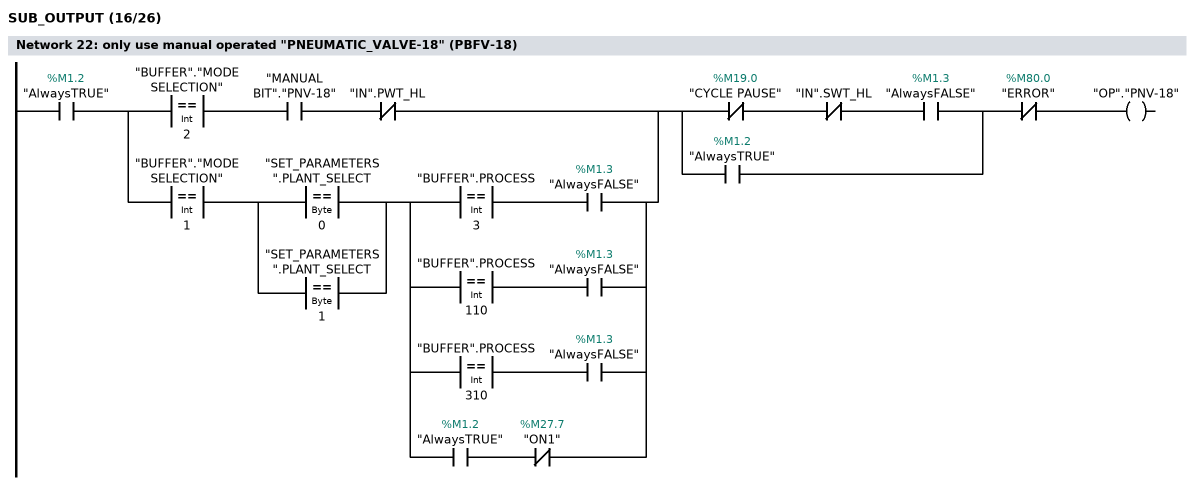
   RUNG wire#powerrail
      Contact( "AlwaysTRUE" )
      wire#w1
      { S7_Templates := "SrcType := Int" } EQ_Contact(in1 := "BUFFER"."MODE SELECTION", in2 := 2)
      Contact( "MANUAL BIT"."PNV-18" )
      I_Contact( "IN".PWT_HL )
      wire#w2
      I_Contact( "CYCLE PAUSE" )
      I_Contact( "IN".SWT_HL )
      Contact( "AlwaysFALSE" )
      wire#w5
      I_Contact( "ERROR" )
      Coil( "OP"."PNV-18" )
   END_RUNG
   RUNG wire#w1
      { S7_Templates := "SrcType := Int" } EQ_Contact(in1 := "BUFFER"."MODE SELECTION", in2 := 1)
      wire#w3
      { S7_Templates := "SrcType := Byte" } EQ_Contact(in1 := "SET_PARAMETERS".PLANT_SELECT, in2 := 0)
      wire#w4
      { S7_Templates := "SrcType := Int" } EQ_Contact(in1 := "BUFFER".PROCESS, in2 := 3)
      Contact( "AlwaysFALSE" )
   END_RUNG wire#w2
   RUNG wire#w3
      { S7_Templates := "SrcType := Byte" } EQ_Contact(in1 := "SET_PARAMETERS".PLANT_SELECT, in2 := 1)
   END_RUNG wire#w4
   RUNG wire#w4
      { S7_Templates := "SrcType := Int" } EQ_Contact(in1 := "BUFFER".PROCESS, in2 := 110)
      Contact( "AlwaysFALSE" )
   END_RUNG wire#w2
   RUNG wire#w4
      { S7_Templates := "SrcType := Int" } EQ_Contact(in1 := "BUFFER".PROCESS, in2 := 310)
      Contact( "AlwaysFALSE" )
   END_RUNG wire#w2
   RUNG wire#w4
      Contact( "AlwaysTRUE" )
      I_Contact( "ON1" )
   END_RUNG wire#w2
   RUNG wire#w2
      Contact( "AlwaysTRUE" )
   END_RUNG wire#w5
   // the same network as SCL:
   "OP"."PNV-18" := "AlwaysTRUE" AND ((("BUFFER"."MODE SELECTION" = 2) AND "MANUAL BIT"."PNV-18" AND NOT "IN".PWT_HL) OR (("BUFFER"."MODE SELECTION" = 1) AND (("SET_PARAMETERS".PLANT_SELECT = 0) OR ("SET_PARAMETERS".PLANT_SELECT = 1)) AND ((("BUFFER".PROCESS = 3) AND "AlwaysFALSE") OR (("BUFFER".PROCESS = 110) AND "AlwaysFALSE") OR (("BUFFER".PROCESS = 310) AND "AlwaysFALSE") OR ("AlwaysTRUE" AND NOT "ON1")))) AND ((NOT "CYCLE PAUSE" AND NOT "IN".SWT_HL AND "AlwaysFALSE") OR "AlwaysTRUE") AND NOT "ERROR";
END_REGION

REGION Network 23: "PNEUMATIC_VALVE-19" (PBFV-19) MFG2 - MFG
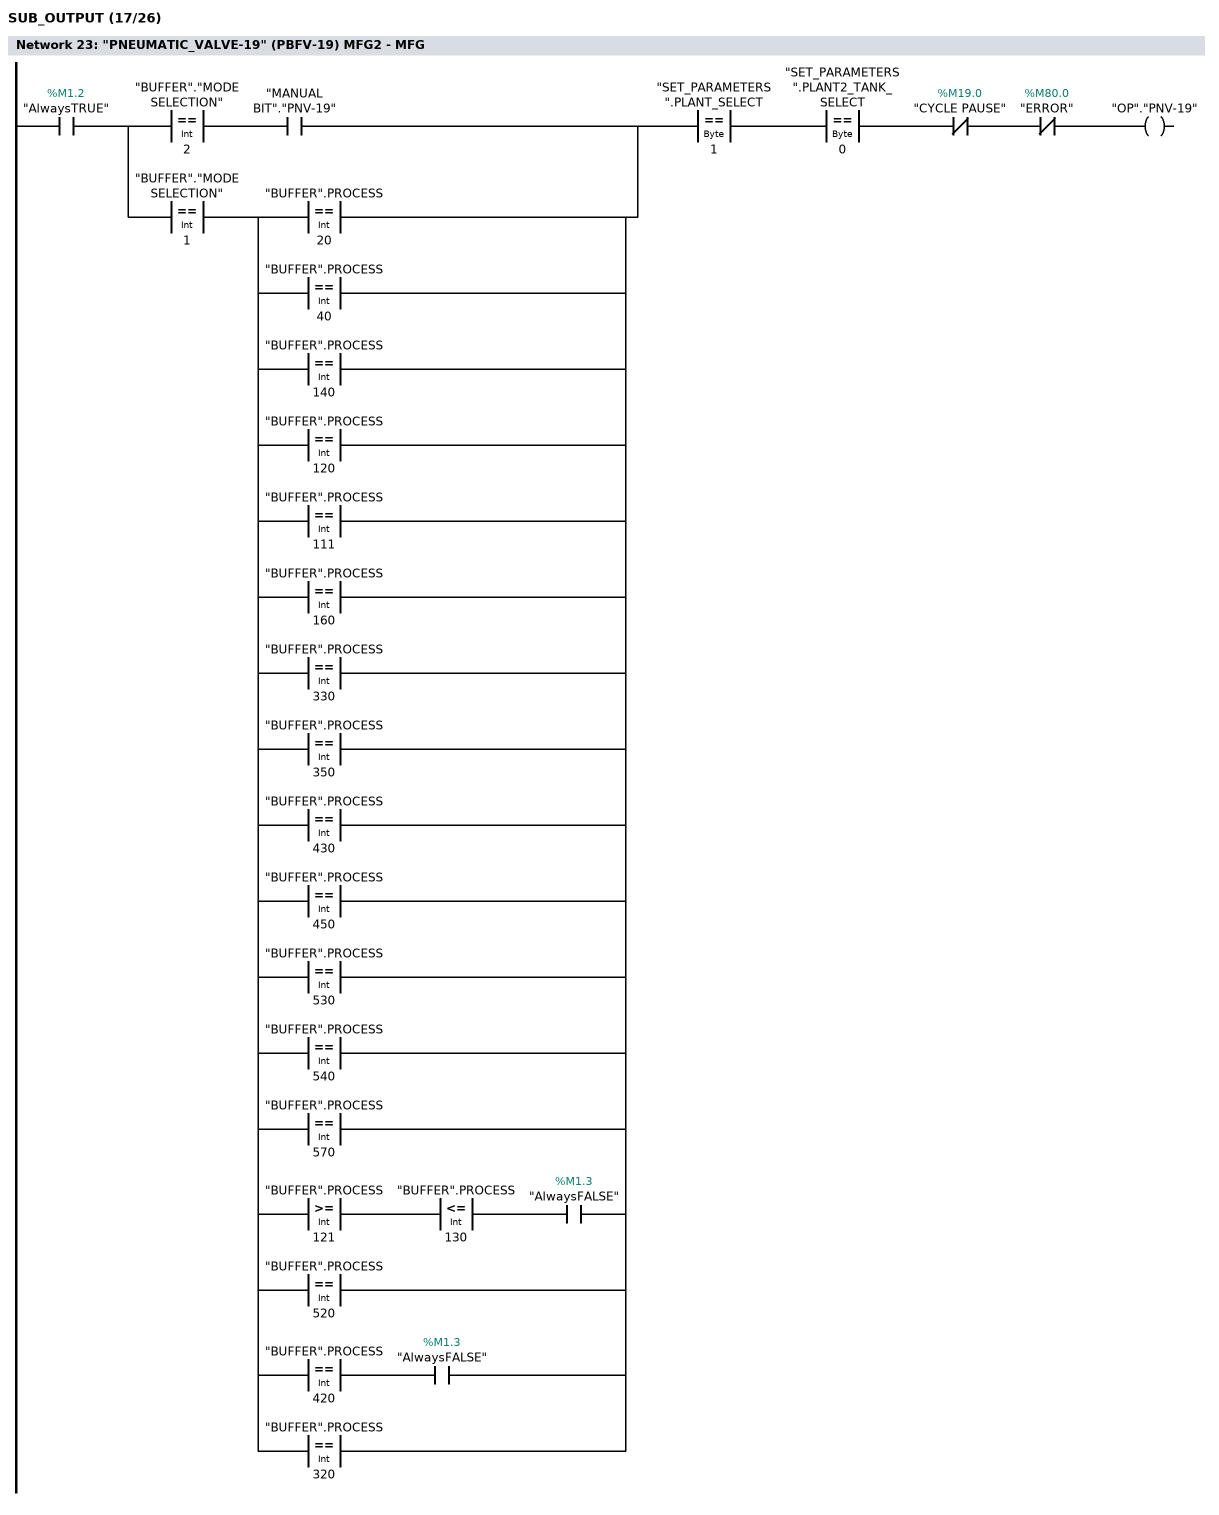
   RUNG wire#powerrail
      Contact( "AlwaysTRUE" )
      wire#w1
      { S7_Templates := "SrcType := Int" } EQ_Contact(in1 := "BUFFER"."MODE SELECTION", in2 := 2)
      Contact( "MANUAL BIT"."PNV-19" )
      wire#w2
      { S7_Templates := "SrcType := Byte" } EQ_Contact(in1 := "SET_PARAMETERS".PLANT_SELECT, in2 := 1)
      { S7_Templates := "SrcType := Byte" } EQ_Contact(in1 := "SET_PARAMETERS".PLANT2_TANK_SELECT, in2 := 0)
      I_Contact( "CYCLE PAUSE" )
      I_Contact( "ERROR" )
      Coil( "OP"."PNV-19" )
   END_RUNG
   RUNG wire#w1
      { S7_Templates := "SrcType := Int" } EQ_Contact(in1 := "BUFFER"."MODE SELECTION", in2 := 1)
      wire#w3
      { S7_Templates := "SrcType := Int" } EQ_Contact(in1 := "BUFFER".PROCESS, in2 := 20)
   END_RUNG wire#w2
   RUNG wire#w3
      { S7_Templates := "SrcType := Int" } EQ_Contact(in1 := "BUFFER".PROCESS, in2 := 40)
   END_RUNG wire#w2
   RUNG wire#w3
      { S7_Templates := "SrcType := Int" } EQ_Contact(in1 := "BUFFER".PROCESS, in2 := 140)
   END_RUNG wire#w2
   RUNG wire#w3
      { S7_Templates := "SrcType := Int" } EQ_Contact(in1 := "BUFFER".PROCESS, in2 := 120)
   END_RUNG wire#w2
   RUNG wire#w3
      { S7_Templates := "SrcType := Int" } EQ_Contact(in1 := "BUFFER".PROCESS, in2 := 111)
   END_RUNG wire#w2
   RUNG wire#w3
      { S7_Templates := "SrcType := Int" } EQ_Contact(in1 := "BUFFER".PROCESS, in2 := 160)
   END_RUNG wire#w2
   RUNG wire#w3
      { S7_Templates := "SrcType := Int" } EQ_Contact(in1 := "BUFFER".PROCESS, in2 := 330)
   END_RUNG wire#w2
   RUNG wire#w3
      { S7_Templates := "SrcType := Int" } EQ_Contact(in1 := "BUFFER".PROCESS, in2 := 350)
   END_RUNG wire#w2
   RUNG wire#w3
      { S7_Templates := "SrcType := Int" } EQ_Contact(in1 := "BUFFER".PROCESS, in2 := 430)
   END_RUNG wire#w2
   RUNG wire#w3
      { S7_Templates := "SrcType := Int" } EQ_Contact(in1 := "BUFFER".PROCESS, in2 := 450)
   END_RUNG wire#w2
   RUNG wire#w3
      { S7_Templates := "SrcType := Int" } EQ_Contact(in1 := "BUFFER".PROCESS, in2 := 530)
   END_RUNG wire#w2
   RUNG wire#w3
      { S7_Templates := "SrcType := Int" } EQ_Contact(in1 := "BUFFER".PROCESS, in2 := 540)
   END_RUNG wire#w2
   RUNG wire#w3
      { S7_Templates := "SrcType := Int" } EQ_Contact(in1 := "BUFFER".PROCESS, in2 := 570)
   END_RUNG wire#w2
   RUNG wire#w3
      { S7_Templates := "SrcType := Int" } GE_Contact(in1 := "BUFFER".PROCESS, in2 := 121)
      { S7_Templates := "SrcType := Int" } LE_Contact(in1 := "BUFFER".PROCESS, in2 := 130)
      Contact( "AlwaysFALSE" )
   END_RUNG wire#w2
   RUNG wire#w3
      { S7_Templates := "SrcType := Int" } EQ_Contact(in1 := "BUFFER".PROCESS, in2 := 520)
   END_RUNG wire#w2
   RUNG wire#w3
      { S7_Templates := "SrcType := Int" } EQ_Contact(in1 := "BUFFER".PROCESS, in2 := 420)
      Contact( "AlwaysFALSE" )
   END_RUNG wire#w2
   RUNG wire#w3
      { S7_Templates := "SrcType := Int" } EQ_Contact(in1 := "BUFFER".PROCESS, in2 := 320)
   END_RUNG wire#w2
   // the same network as SCL:
   "OP"."PNV-19" := "AlwaysTRUE" AND ((("BUFFER"."MODE SELECTION" = 2) AND "MANUAL BIT"."PNV-19") OR (("BUFFER"."MODE SELECTION" = 1) AND (("BUFFER".PROCESS = 20) OR ("BUFFER".PROCESS = 40) OR ("BUFFER".PROCESS = 140) OR ("BUFFER".PROCESS = 120) OR ("BUFFER".PROCESS = 111) OR ("BUFFER".PROCESS = 160) OR ("BUFFER".PROCESS = 330) OR ("BUFFER".PROCESS = 350) OR ("BUFFER".PROCESS = 430) OR ("BUFFER".PROCESS = 450) OR ("BUFFER".PROCESS = 530) OR ("BUFFER".PROCESS = 540) OR ("BUFFER".PROCESS = 570) OR (("BUFFER".PROCESS >= 121) AND ("BUFFER".PROCESS <= 130) AND "AlwaysFALSE") OR ("BUFFER".PROCESS = 520) OR (("BUFFER".PROCESS = 420) AND "AlwaysFALSE") OR ("BUFFER".PROCESS = 320)))) AND ("SET_PARAMETERS".PLANT_SELECT = 1) AND ("SET_PARAMETERS".PLANT2_TANK_SELECT = 0) AND NOT "CYCLE PAUSE" AND NOT "ERROR";
END_REGION

REGION Network 24: "PNEUMATIC_VALVE-20" (PBFV-20) MFG2- STORAGE1
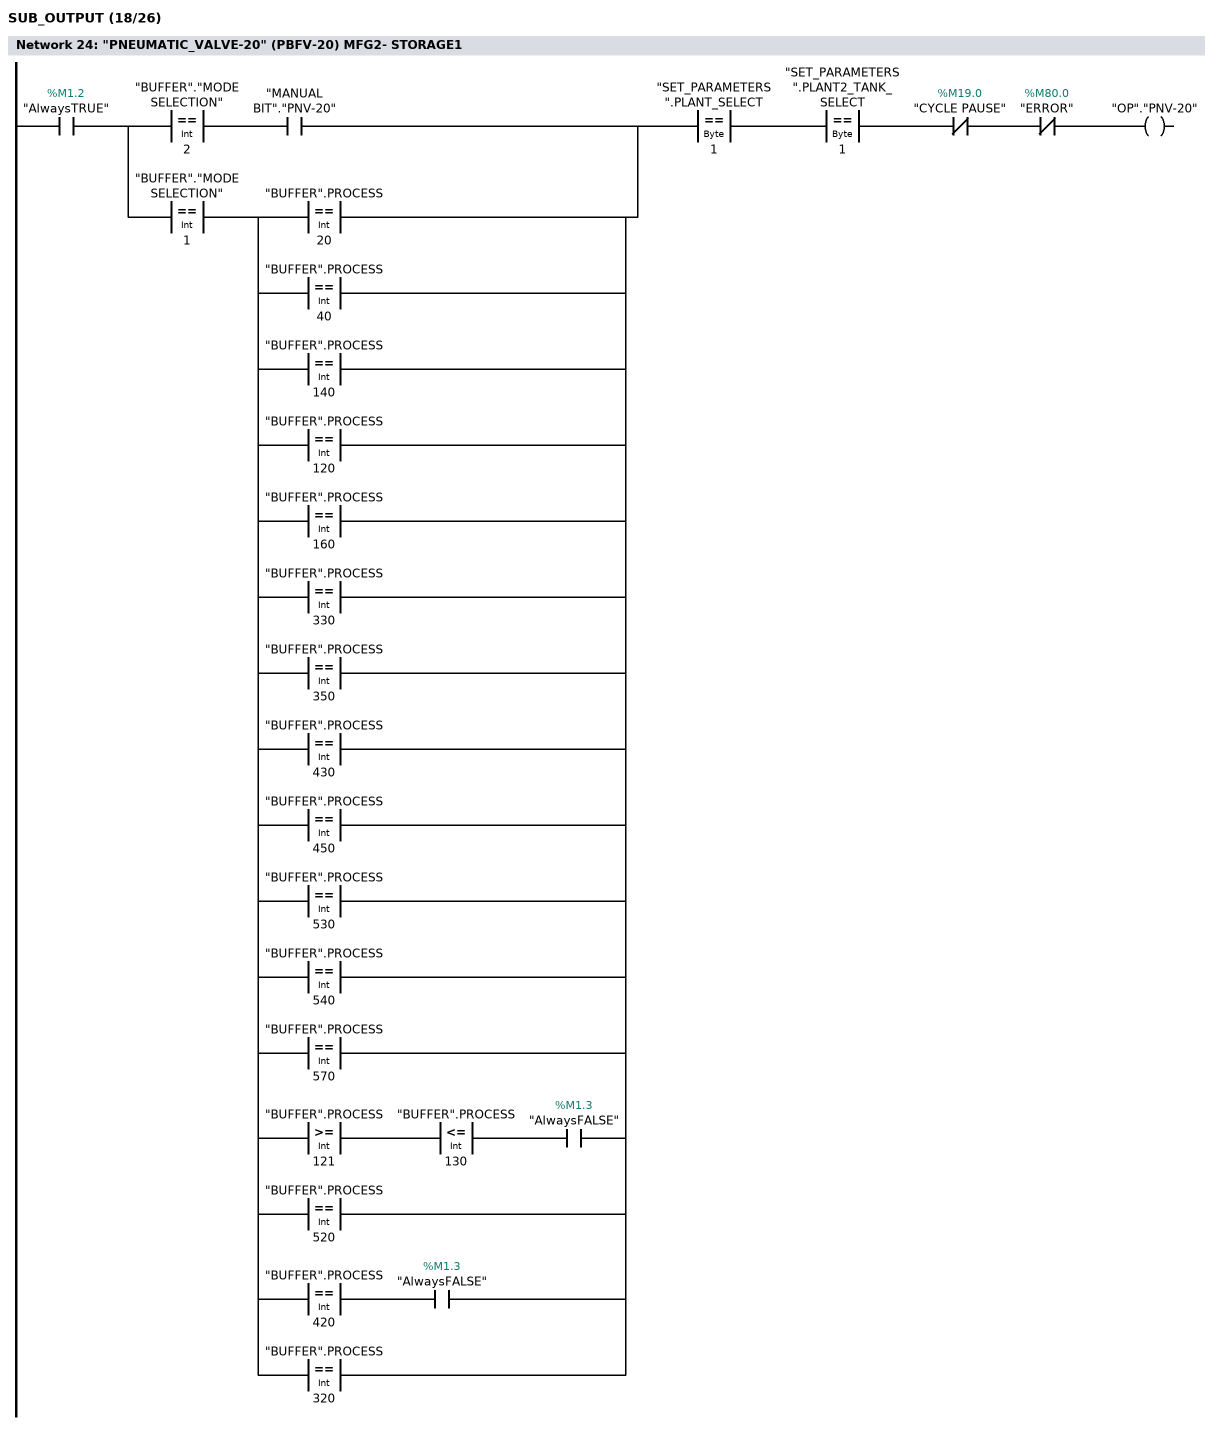
   RUNG wire#powerrail
      Contact( "AlwaysTRUE" )
      wire#w1
      { S7_Templates := "SrcType := Int" } EQ_Contact(in1 := "BUFFER"."MODE SELECTION", in2 := 2)
      Contact( "MANUAL BIT"."PNV-20" )
      wire#w2
      { S7_Templates := "SrcType := Byte" } EQ_Contact(in1 := "SET_PARAMETERS".PLANT_SELECT, in2 := 1)
      { S7_Templates := "SrcType := Byte" } EQ_Contact(in1 := "SET_PARAMETERS".PLANT2_TANK_SELECT, in2 := 1)
      I_Contact( "CYCLE PAUSE" )
      I_Contact( "ERROR" )
      Coil( "OP"."PNV-20" )
   END_RUNG
   RUNG wire#w1
      { S7_Templates := "SrcType := Int" } EQ_Contact(in1 := "BUFFER"."MODE SELECTION", in2 := 1)
      wire#w3
      { S7_Templates := "SrcType := Int" } EQ_Contact(in1 := "BUFFER".PROCESS, in2 := 20)
   END_RUNG wire#w2
   RUNG wire#w3
      { S7_Templates := "SrcType := Int" } EQ_Contact(in1 := "BUFFER".PROCESS, in2 := 40)
   END_RUNG wire#w2
   RUNG wire#w3
      { S7_Templates := "SrcType := Int" } EQ_Contact(in1 := "BUFFER".PROCESS, in2 := 140)
   END_RUNG wire#w2
   RUNG wire#w3
      { S7_Templates := "SrcType := Int" } EQ_Contact(in1 := "BUFFER".PROCESS, in2 := 120)
   END_RUNG wire#w2
   RUNG wire#w3
      { S7_Templates := "SrcType := Int" } EQ_Contact(in1 := "BUFFER".PROCESS, in2 := 160)
   END_RUNG wire#w2
   RUNG wire#w3
      { S7_Templates := "SrcType := Int" } EQ_Contact(in1 := "BUFFER".PROCESS, in2 := 330)
   END_RUNG wire#w2
   RUNG wire#w3
      { S7_Templates := "SrcType := Int" } EQ_Contact(in1 := "BUFFER".PROCESS, in2 := 350)
   END_RUNG wire#w2
   RUNG wire#w3
      { S7_Templates := "SrcType := Int" } EQ_Contact(in1 := "BUFFER".PROCESS, in2 := 430)
   END_RUNG wire#w2
   RUNG wire#w3
      { S7_Templates := "SrcType := Int" } EQ_Contact(in1 := "BUFFER".PROCESS, in2 := 450)
   END_RUNG wire#w2
   RUNG wire#w3
      { S7_Templates := "SrcType := Int" } EQ_Contact(in1 := "BUFFER".PROCESS, in2 := 530)
   END_RUNG wire#w2
   RUNG wire#w3
      { S7_Templates := "SrcType := Int" } EQ_Contact(in1 := "BUFFER".PROCESS, in2 := 540)
   END_RUNG wire#w2
   RUNG wire#w3
      { S7_Templates := "SrcType := Int" } EQ_Contact(in1 := "BUFFER".PROCESS, in2 := 570)
   END_RUNG wire#w2
   RUNG wire#w3
      { S7_Templates := "SrcType := Int" } GE_Contact(in1 := "BUFFER".PROCESS, in2 := 121)
      { S7_Templates := "SrcType := Int" } LE_Contact(in1 := "BUFFER".PROCESS, in2 := 130)
      Contact( "AlwaysFALSE" )
   END_RUNG wire#w2
   RUNG wire#w3
      { S7_Templates := "SrcType := Int" } EQ_Contact(in1 := "BUFFER".PROCESS, in2 := 520)
   END_RUNG wire#w2
   RUNG wire#w3
      { S7_Templates := "SrcType := Int" } EQ_Contact(in1 := "BUFFER".PROCESS, in2 := 420)
      Contact( "AlwaysFALSE" )
   END_RUNG wire#w2
   RUNG wire#w3
      { S7_Templates := "SrcType := Int" } EQ_Contact(in1 := "BUFFER".PROCESS, in2 := 320)
   END_RUNG wire#w2
   // the same network as SCL:
   "OP"."PNV-20" := "AlwaysTRUE" AND ((("BUFFER"."MODE SELECTION" = 2) AND "MANUAL BIT"."PNV-20") OR (("BUFFER"."MODE SELECTION" = 1) AND (("BUFFER".PROCESS = 20) OR ("BUFFER".PROCESS = 40) OR ("BUFFER".PROCESS = 140) OR ("BUFFER".PROCESS = 120) OR ("BUFFER".PROCESS = 160) OR ("BUFFER".PROCESS = 330) OR ("BUFFER".PROCESS = 350) OR ("BUFFER".PROCESS = 430) OR ("BUFFER".PROCESS = 450) OR ("BUFFER".PROCESS = 530) OR ("BUFFER".PROCESS = 540) OR ("BUFFER".PROCESS = 570) OR (("BUFFER".PROCESS >= 121) AND ("BUFFER".PROCESS <= 130) AND "AlwaysFALSE") OR ("BUFFER".PROCESS = 520) OR (("BUFFER".PROCESS = 420) AND "AlwaysFALSE") OR ("BUFFER".PROCESS = 320)))) AND ("SET_PARAMETERS".PLANT_SELECT = 1) AND ("SET_PARAMETERS".PLANT2_TANK_SELECT = 1) AND NOT "CYCLE PAUSE" AND NOT "ERROR";
END_REGION

REGION Network 25: "PNEUMATIC_VALVE-21" (PV-21)
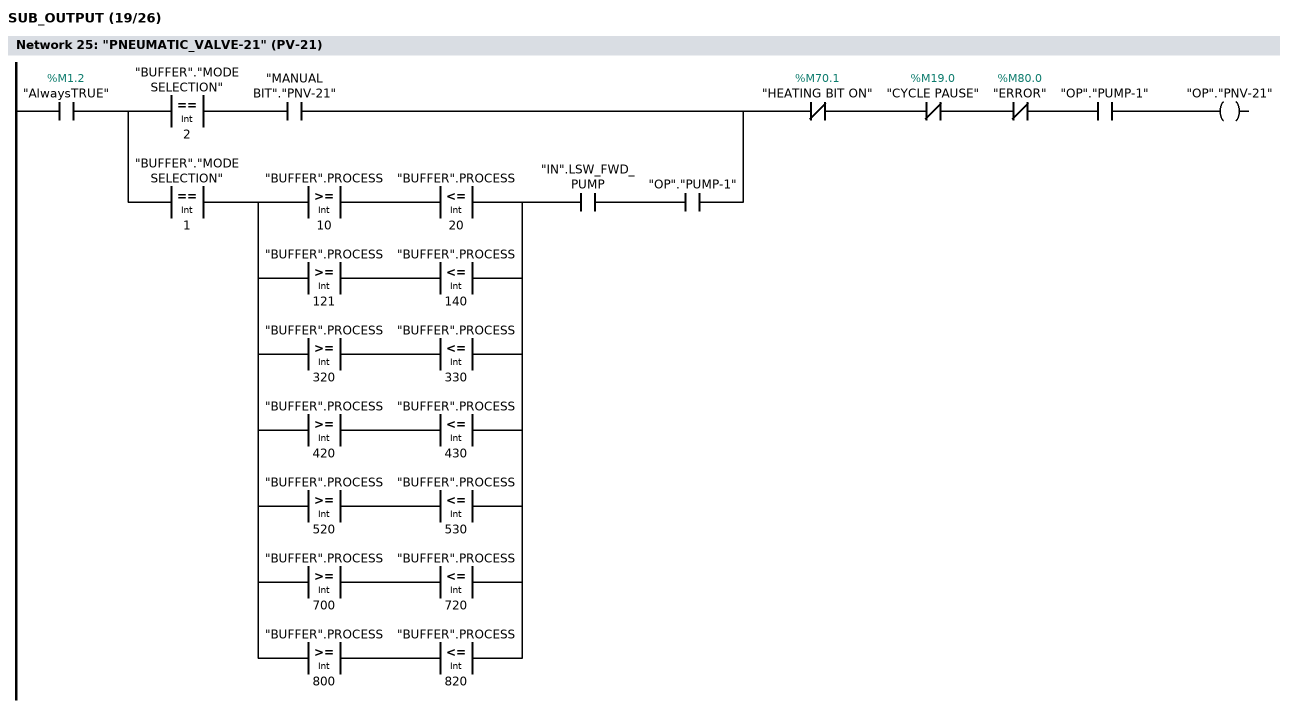
   RUNG wire#powerrail
      Contact( "AlwaysTRUE" )
      wire#w1
      { S7_Templates := "SrcType := Int" } EQ_Contact(in1 := "BUFFER"."MODE SELECTION", in2 := 2)
      Contact( "MANUAL BIT"."PNV-21" )
      wire#w2
      I_Contact( "HEATING BIT ON" )
      I_Contact( "CYCLE PAUSE" )
      I_Contact( "ERROR" )
      Contact( "OP"."PUMP-1" )
      Coil( "OP"."PNV-21" )
   END_RUNG
   RUNG wire#w1
      { S7_Templates := "SrcType := Int" } EQ_Contact(in1 := "BUFFER"."MODE SELECTION", in2 := 1)
      wire#w3
      { S7_Templates := "SrcType := Int" } GE_Contact(in1 := "BUFFER".PROCESS, in2 := 10)
      { S7_Templates := "SrcType := Int" } LE_Contact(in1 := "BUFFER".PROCESS, in2 := 20)
      wire#w4
      Contact( "IN".LSW_FWD_PUMP )
      Contact( "OP"."PUMP-1" )
   END_RUNG wire#w2
   RUNG wire#w3
      { S7_Templates := "SrcType := Int" } GE_Contact(in1 := "BUFFER".PROCESS, in2 := 121)
      { S7_Templates := "SrcType := Int" } LE_Contact(in1 := "BUFFER".PROCESS, in2 := 140)
   END_RUNG wire#w4
   RUNG wire#w3
      { S7_Templates := "SrcType := Int" } GE_Contact(in1 := "BUFFER".PROCESS, in2 := 320)
      { S7_Templates := "SrcType := Int" } LE_Contact(in1 := "BUFFER".PROCESS, in2 := 330)
   END_RUNG wire#w4
   RUNG wire#w3
      { S7_Templates := "SrcType := Int" } GE_Contact(in1 := "BUFFER".PROCESS, in2 := 420)
      { S7_Templates := "SrcType := Int" } LE_Contact(in1 := "BUFFER".PROCESS, in2 := 430)
   END_RUNG wire#w4
   RUNG wire#w3
      { S7_Templates := "SrcType := Int" } GE_Contact(in1 := "BUFFER".PROCESS, in2 := 520)
      { S7_Templates := "SrcType := Int" } LE_Contact(in1 := "BUFFER".PROCESS, in2 := 530)
   END_RUNG wire#w4
   RUNG wire#w3
      { S7_Templates := "SrcType := Int" } GE_Contact(in1 := "BUFFER".PROCESS, in2 := 700)
      { S7_Templates := "SrcType := Int" } LE_Contact(in1 := "BUFFER".PROCESS, in2 := 720)
   END_RUNG wire#w4
   RUNG wire#w3
      { S7_Templates := "SrcType := Int" } GE_Contact(in1 := "BUFFER".PROCESS, in2 := 800)
      { S7_Templates := "SrcType := Int" } LE_Contact(in1 := "BUFFER".PROCESS, in2 := 820)
   END_RUNG wire#w4
   // the same network as SCL:
   "OP"."PNV-21" := "AlwaysTRUE" AND ((("BUFFER"."MODE SELECTION" = 2) AND "MANUAL BIT"."PNV-21") OR (("BUFFER"."MODE SELECTION" = 1) AND ((("BUFFER".PROCESS >= 10) AND ("BUFFER".PROCESS <= 20)) OR (("BUFFER".PROCESS >= 121) AND ("BUFFER".PROCESS <= 140)) OR (("BUFFER".PROCESS >= 320) AND ("BUFFER".PROCESS <= 330)) OR (("BUFFER".PROCESS >= 420) AND ("BUFFER".PROCESS <= 430)) OR (("BUFFER".PROCESS >= 520) AND ("BUFFER".PROCESS <= 530)) OR (("BUFFER".PROCESS >= 700) AND ("BUFFER".PROCESS <= 720)) OR (("BUFFER".PROCESS >= 800) AND ("BUFFER".PROCESS <= 820))) AND "IN".LSW_FWD_PUMP AND "OP"."PUMP-1")) AND NOT "HEATING BIT ON" AND NOT "CYCLE PAUSE" AND NOT "ERROR" AND "OP"."PUMP-1";
END_REGION

REGION Network 26: "PNEUMATIC_VALVE-22" (PV-22)
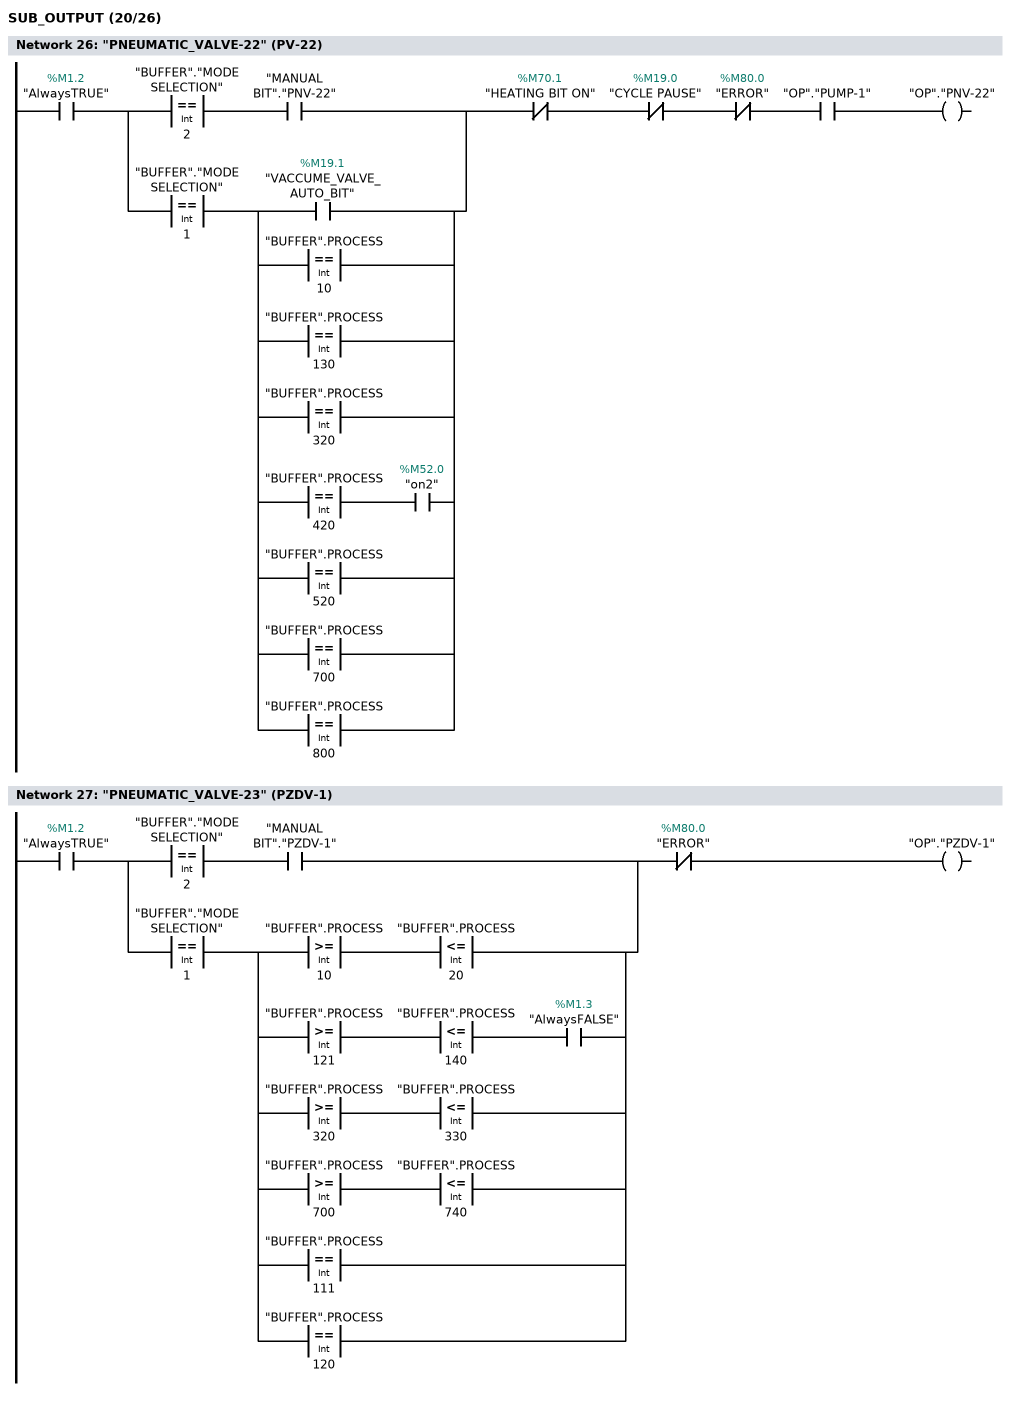
   RUNG wire#powerrail
      Contact( "AlwaysTRUE" )
      wire#w1
      { S7_Templates := "SrcType := Int" } EQ_Contact(in1 := "BUFFER"."MODE SELECTION", in2 := 2)
      Contact( "MANUAL BIT"."PNV-22" )
      wire#w2
      I_Contact( "HEATING BIT ON" )
      I_Contact( "CYCLE PAUSE" )
      I_Contact( "ERROR" )
      Contact( "OP"."PUMP-1" )
      Coil( "OP"."PNV-22" )
   END_RUNG
   RUNG wire#w1
      { S7_Templates := "SrcType := Int" } EQ_Contact(in1 := "BUFFER"."MODE SELECTION", in2 := 1)
      wire#w3
      Contact( "VACCUME_VALVE_AUTO_BIT" )
   END_RUNG wire#w2
   RUNG wire#w3
      { S7_Templates := "SrcType := Int" } EQ_Contact(in1 := "BUFFER".PROCESS, in2 := 10)
   END_RUNG wire#w2
   RUNG wire#w3
      { S7_Templates := "SrcType := Int" } EQ_Contact(in1 := "BUFFER".PROCESS, in2 := 130)
   END_RUNG wire#w2
   RUNG wire#w3
      { S7_Templates := "SrcType := Int" } EQ_Contact(in1 := "BUFFER".PROCESS, in2 := 320)
   END_RUNG wire#w2
   RUNG wire#w3
      { S7_Templates := "SrcType := Int" } EQ_Contact(in1 := "BUFFER".PROCESS, in2 := 420)
      Contact( "on2" )
   END_RUNG wire#w2
   RUNG wire#w3
      { S7_Templates := "SrcType := Int" } EQ_Contact(in1 := "BUFFER".PROCESS, in2 := 520)
   END_RUNG wire#w2
   RUNG wire#w3
      { S7_Templates := "SrcType := Int" } EQ_Contact(in1 := "BUFFER".PROCESS, in2 := 700)
   END_RUNG wire#w2
   RUNG wire#w3
      { S7_Templates := "SrcType := Int" } EQ_Contact(in1 := "BUFFER".PROCESS, in2 := 800)
   END_RUNG wire#w2
   // the same network as SCL:
   "OP"."PNV-22" := "AlwaysTRUE" AND ((("BUFFER"."MODE SELECTION" = 2) AND "MANUAL BIT"."PNV-22") OR (("BUFFER"."MODE SELECTION" = 1) AND ("VACCUME_VALVE_AUTO_BIT" OR ("BUFFER".PROCESS = 10) OR ("BUFFER".PROCESS = 130) OR ("BUFFER".PROCESS = 320) OR (("BUFFER".PROCESS = 420) AND "on2") OR ("BUFFER".PROCESS = 520) OR ("BUFFER".PROCESS = 700) OR ("BUFFER".PROCESS = 800)))) AND NOT "HEATING BIT ON" AND NOT "CYCLE PAUSE" AND NOT "ERROR" AND "OP"."PUMP-1";
END_REGION

REGION Network 27: "PNEUMATIC_VALVE-23" (PZDV-1)
   RUNG wire#powerrail
      Contact( "AlwaysTRUE" )
      wire#w1
      { S7_Templates := "SrcType := Int" } EQ_Contact(in1 := "BUFFER"."MODE SELECTION", in2 := 2)
      Contact( "MANUAL BIT"."PZDV-1" )
      wire#w2
      I_Contact( "ERROR" )
      Coil( "OP"."PZDV-1" )
   END_RUNG
   RUNG wire#w1
      { S7_Templates := "SrcType := Int" } EQ_Contact(in1 := "BUFFER"."MODE SELECTION", in2 := 1)
      wire#w3
      { S7_Templates := "SrcType := Int" } GE_Contact(in1 := "BUFFER".PROCESS, in2 := 10)
      { S7_Templates := "SrcType := Int" } LE_Contact(in1 := "BUFFER".PROCESS, in2 := 20)
   END_RUNG wire#w2
   RUNG wire#w3
      { S7_Templates := "SrcType := Int" } GE_Contact(in1 := "BUFFER".PROCESS, in2 := 121)
      { S7_Templates := "SrcType := Int" } LE_Contact(in1 := "BUFFER".PROCESS, in2 := 140)
      Contact( "AlwaysFALSE" )
   END_RUNG wire#w2
   RUNG wire#w3
      { S7_Templates := "SrcType := Int" } GE_Contact(in1 := "BUFFER".PROCESS, in2 := 320)
      { S7_Templates := "SrcType := Int" } LE_Contact(in1 := "BUFFER".PROCESS, in2 := 330)
   END_RUNG wire#w2
   RUNG wire#w3
      { S7_Templates := "SrcType := Int" } GE_Contact(in1 := "BUFFER".PROCESS, in2 := 700)
      { S7_Templates := "SrcType := Int" } LE_Contact(in1 := "BUFFER".PROCESS, in2 := 740)
   END_RUNG wire#w2
   RUNG wire#w3
      { S7_Templates := "SrcType := Int" } EQ_Contact(in1 := "BUFFER".PROCESS, in2 := 111)
   END_RUNG wire#w2
   RUNG wire#w3
      { S7_Templates := "SrcType := Int" } EQ_Contact(in1 := "BUFFER".PROCESS, in2 := 120)
   END_RUNG wire#w2
   // the same network as SCL:
   "OP"."PZDV-1" := "AlwaysTRUE" AND ((("BUFFER"."MODE SELECTION" = 2) AND "MANUAL BIT"."PZDV-1") OR (("BUFFER"."MODE SELECTION" = 1) AND ((("BUFFER".PROCESS >= 10) AND ("BUFFER".PROCESS <= 20)) OR (("BUFFER".PROCESS >= 121) AND ("BUFFER".PROCESS <= 140) AND "AlwaysFALSE") OR (("BUFFER".PROCESS >= 320) AND ("BUFFER".PROCESS <= 330)) OR (("BUFFER".PROCESS >= 700) AND ("BUFFER".PROCESS <= 740)) OR ("BUFFER".PROCESS = 111) OR ("BUFFER".PROCESS = 120)))) AND NOT "ERROR";
END_REGION

REGION Network 28: "PNEUMATIC_VALVE-24" (PZDV-2)
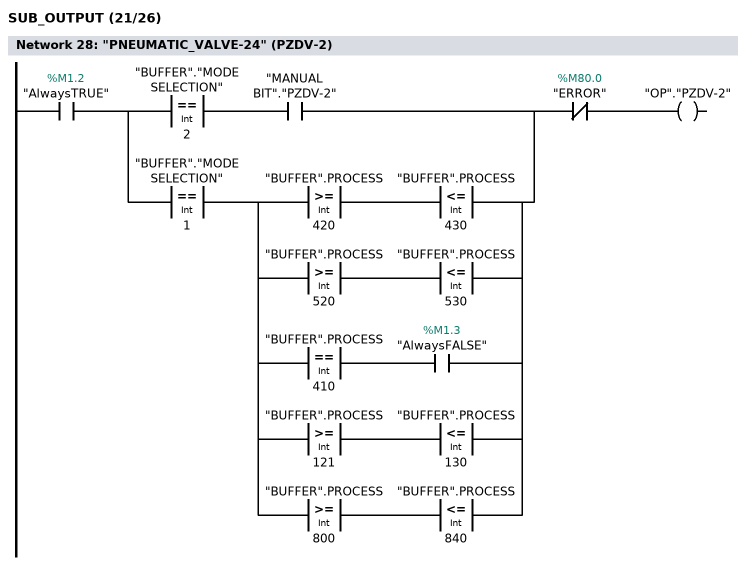
   RUNG wire#powerrail
      Contact( "AlwaysTRUE" )
      wire#w1
      { S7_Templates := "SrcType := Int" } EQ_Contact(in1 := "BUFFER"."MODE SELECTION", in2 := 2)
      Contact( "MANUAL BIT"."PZDV-2" )
      wire#w2
      I_Contact( "ERROR" )
      Coil( "OP"."PZDV-2" )
   END_RUNG
   RUNG wire#w1
      { S7_Templates := "SrcType := Int" } EQ_Contact(in1 := "BUFFER"."MODE SELECTION", in2 := 1)
      wire#w3
      { S7_Templates := "SrcType := Int" } GE_Contact(in1 := "BUFFER".PROCESS, in2 := 420)
      { S7_Templates := "SrcType := Int" } LE_Contact(in1 := "BUFFER".PROCESS, in2 := 430)
   END_RUNG wire#w2
   RUNG wire#w3
      { S7_Templates := "SrcType := Int" } GE_Contact(in1 := "BUFFER".PROCESS, in2 := 520)
      { S7_Templates := "SrcType := Int" } LE_Contact(in1 := "BUFFER".PROCESS, in2 := 530)
   END_RUNG wire#w2
   RUNG wire#w3
      { S7_Templates := "SrcType := Int" } EQ_Contact(in1 := "BUFFER".PROCESS, in2 := 410)
      Contact( "AlwaysFALSE" )
   END_RUNG wire#w2
   RUNG wire#w3
      { S7_Templates := "SrcType := Int" } GE_Contact(in1 := "BUFFER".PROCESS, in2 := 121)
      { S7_Templates := "SrcType := Int" } LE_Contact(in1 := "BUFFER".PROCESS, in2 := 130)
   END_RUNG wire#w2
   RUNG wire#w3
      { S7_Templates := "SrcType := Int" } GE_Contact(in1 := "BUFFER".PROCESS, in2 := 800)
      { S7_Templates := "SrcType := Int" } LE_Contact(in1 := "BUFFER".PROCESS, in2 := 840)
   END_RUNG wire#w2
   // the same network as SCL:
   "OP"."PZDV-2" := "AlwaysTRUE" AND ((("BUFFER"."MODE SELECTION" = 2) AND "MANUAL BIT"."PZDV-2") OR (("BUFFER"."MODE SELECTION" = 1) AND ((("BUFFER".PROCESS >= 420) AND ("BUFFER".PROCESS <= 430)) OR (("BUFFER".PROCESS >= 520) AND ("BUFFER".PROCESS <= 530)) OR (("BUFFER".PROCESS = 410) AND "AlwaysFALSE") OR (("BUFFER".PROCESS >= 121) AND ("BUFFER".PROCESS <= 130)) OR (("BUFFER".PROCESS >= 800) AND ("BUFFER".PROCESS <= 840))))) AND NOT "ERROR";
END_REGION

REGION Network 29: "PNEUMATIC_VALVE-25" (CIP_IN) MFG2- STORAGE2 PBFV-23
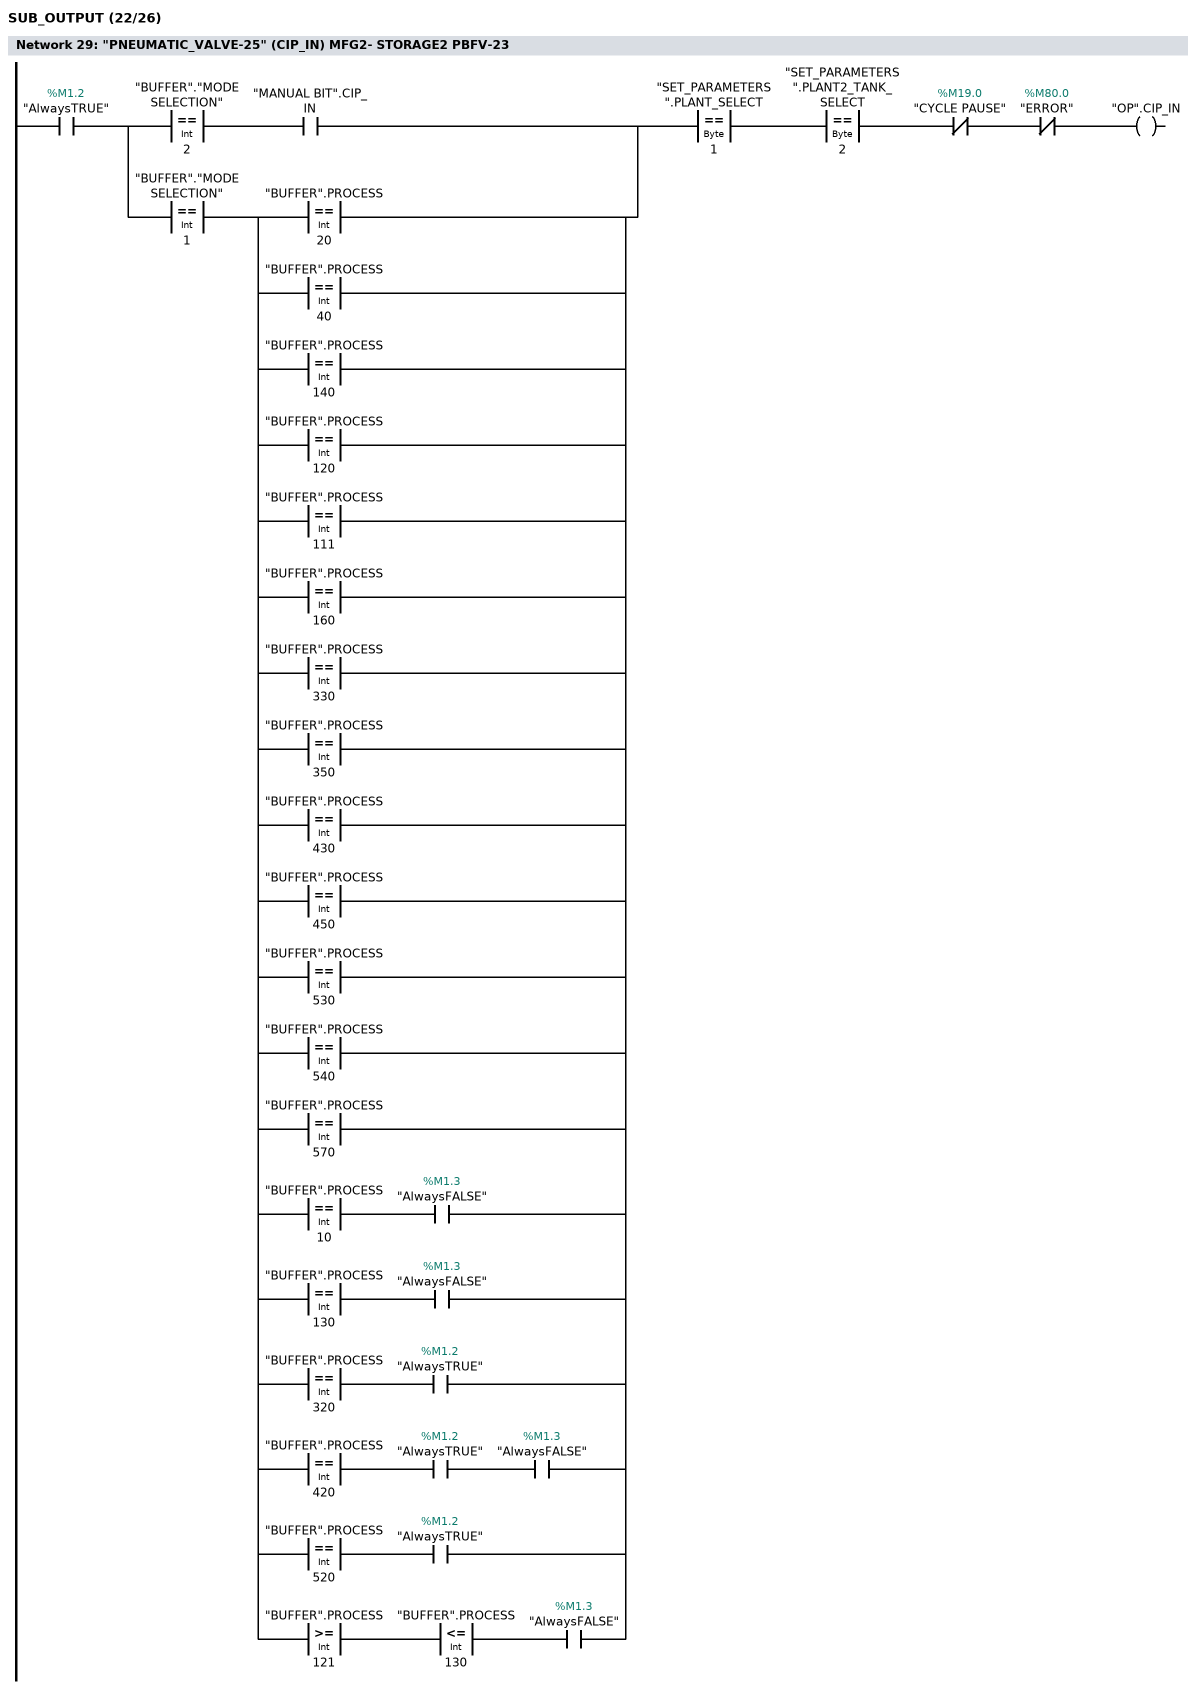
   RUNG wire#powerrail
      Contact( "AlwaysTRUE" )
      wire#w1
      { S7_Templates := "SrcType := Int" } EQ_Contact(in1 := "BUFFER"."MODE SELECTION", in2 := 2)
      Contact( "MANUAL BIT".CIP_IN )
      wire#w2
      { S7_Templates := "SrcType := Byte" } EQ_Contact(in1 := "SET_PARAMETERS".PLANT_SELECT, in2 := 1)
      { S7_Templates := "SrcType := Byte" } EQ_Contact(in1 := "SET_PARAMETERS".PLANT2_TANK_SELECT, in2 := 2)
      I_Contact( "CYCLE PAUSE" )
      I_Contact( "ERROR" )
      Coil( "OP".CIP_IN )
   END_RUNG
   RUNG wire#w1
      { S7_Templates := "SrcType := Int" } EQ_Contact(in1 := "BUFFER"."MODE SELECTION", in2 := 1)
      wire#w3
      { S7_Templates := "SrcType := Int" } EQ_Contact(in1 := "BUFFER".PROCESS, in2 := 20)
   END_RUNG wire#w2
   RUNG wire#w3
      { S7_Templates := "SrcType := Int" } EQ_Contact(in1 := "BUFFER".PROCESS, in2 := 40)
   END_RUNG wire#w2
   RUNG wire#w3
      { S7_Templates := "SrcType := Int" } EQ_Contact(in1 := "BUFFER".PROCESS, in2 := 140)
   END_RUNG wire#w2
   RUNG wire#w3
      { S7_Templates := "SrcType := Int" } EQ_Contact(in1 := "BUFFER".PROCESS, in2 := 120)
   END_RUNG wire#w2
   RUNG wire#w3
      { S7_Templates := "SrcType := Int" } EQ_Contact(in1 := "BUFFER".PROCESS, in2 := 111)
   END_RUNG wire#w2
   RUNG wire#w3
      { S7_Templates := "SrcType := Int" } EQ_Contact(in1 := "BUFFER".PROCESS, in2 := 160)
   END_RUNG wire#w2
   RUNG wire#w3
      { S7_Templates := "SrcType := Int" } EQ_Contact(in1 := "BUFFER".PROCESS, in2 := 330)
   END_RUNG wire#w2
   RUNG wire#w3
      { S7_Templates := "SrcType := Int" } EQ_Contact(in1 := "BUFFER".PROCESS, in2 := 350)
   END_RUNG wire#w2
   RUNG wire#w3
      { S7_Templates := "SrcType := Int" } EQ_Contact(in1 := "BUFFER".PROCESS, in2 := 430)
   END_RUNG wire#w2
   RUNG wire#w3
      { S7_Templates := "SrcType := Int" } EQ_Contact(in1 := "BUFFER".PROCESS, in2 := 450)
   END_RUNG wire#w2
   RUNG wire#w3
      { S7_Templates := "SrcType := Int" } EQ_Contact(in1 := "BUFFER".PROCESS, in2 := 530)
   END_RUNG wire#w2
   RUNG wire#w3
      { S7_Templates := "SrcType := Int" } EQ_Contact(in1 := "BUFFER".PROCESS, in2 := 540)
   END_RUNG wire#w2
   RUNG wire#w3
      { S7_Templates := "SrcType := Int" } EQ_Contact(in1 := "BUFFER".PROCESS, in2 := 570)
   END_RUNG wire#w2
   RUNG wire#w3
      { S7_Templates := "SrcType := Int" } EQ_Contact(in1 := "BUFFER".PROCESS, in2 := 10)
      Contact( "AlwaysFALSE" )
   END_RUNG wire#w2
   RUNG wire#w3
      { S7_Templates := "SrcType := Int" } EQ_Contact(in1 := "BUFFER".PROCESS, in2 := 130)
      Contact( "AlwaysFALSE" )
   END_RUNG wire#w2
   RUNG wire#w3
      { S7_Templates := "SrcType := Int" } EQ_Contact(in1 := "BUFFER".PROCESS, in2 := 320)
      Contact( "AlwaysTRUE" )
   END_RUNG wire#w2
   RUNG wire#w3
      { S7_Templates := "SrcType := Int" } EQ_Contact(in1 := "BUFFER".PROCESS, in2 := 420)
      Contact( "AlwaysTRUE" )
      Contact( "AlwaysFALSE" )
   END_RUNG wire#w2
   RUNG wire#w3
      { S7_Templates := "SrcType := Int" } EQ_Contact(in1 := "BUFFER".PROCESS, in2 := 520)
      Contact( "AlwaysTRUE" )
   END_RUNG wire#w2
   RUNG wire#w3
      { S7_Templates := "SrcType := Int" } GE_Contact(in1 := "BUFFER".PROCESS, in2 := 121)
      { S7_Templates := "SrcType := Int" } LE_Contact(in1 := "BUFFER".PROCESS, in2 := 130)
      Contact( "AlwaysFALSE" )
   END_RUNG wire#w2
   // the same network as SCL:
   "OP".CIP_IN := "AlwaysTRUE" AND ((("BUFFER"."MODE SELECTION" = 2) AND "MANUAL BIT".CIP_IN) OR (("BUFFER"."MODE SELECTION" = 1) AND (("BUFFER".PROCESS = 20) OR ("BUFFER".PROCESS = 40) OR ("BUFFER".PROCESS = 140) OR ("BUFFER".PROCESS = 120) OR ("BUFFER".PROCESS = 111) OR ("BUFFER".PROCESS = 160) OR ("BUFFER".PROCESS = 330) OR ("BUFFER".PROCESS = 350) OR ("BUFFER".PROCESS = 430) OR ("BUFFER".PROCESS = 450) OR ("BUFFER".PROCESS = 530) OR ("BUFFER".PROCESS = 540) OR ("BUFFER".PROCESS = 570) OR (("BUFFER".PROCESS = 10) AND "AlwaysFALSE") OR (("BUFFER".PROCESS = 130) AND "AlwaysFALSE") OR (("BUFFER".PROCESS = 320) AND "AlwaysTRUE") OR (("BUFFER".PROCESS = 420) AND "AlwaysTRUE" AND "AlwaysFALSE") OR (("BUFFER".PROCESS = 520) AND "AlwaysTRUE") OR (("BUFFER".PROCESS >= 121) AND ("BUFFER".PROCESS <= 130) AND "AlwaysFALSE")))) AND ("SET_PARAMETERS".PLANT_SELECT = 1) AND ("SET_PARAMETERS".PLANT2_TANK_SELECT = 2) AND NOT "CYCLE PAUSE" AND NOT "ERROR";
END_REGION

REGION Network 30: "PNEUMATIC_VALVE-26" (CIP_OUT) MFG2- MIXING PBFV-24
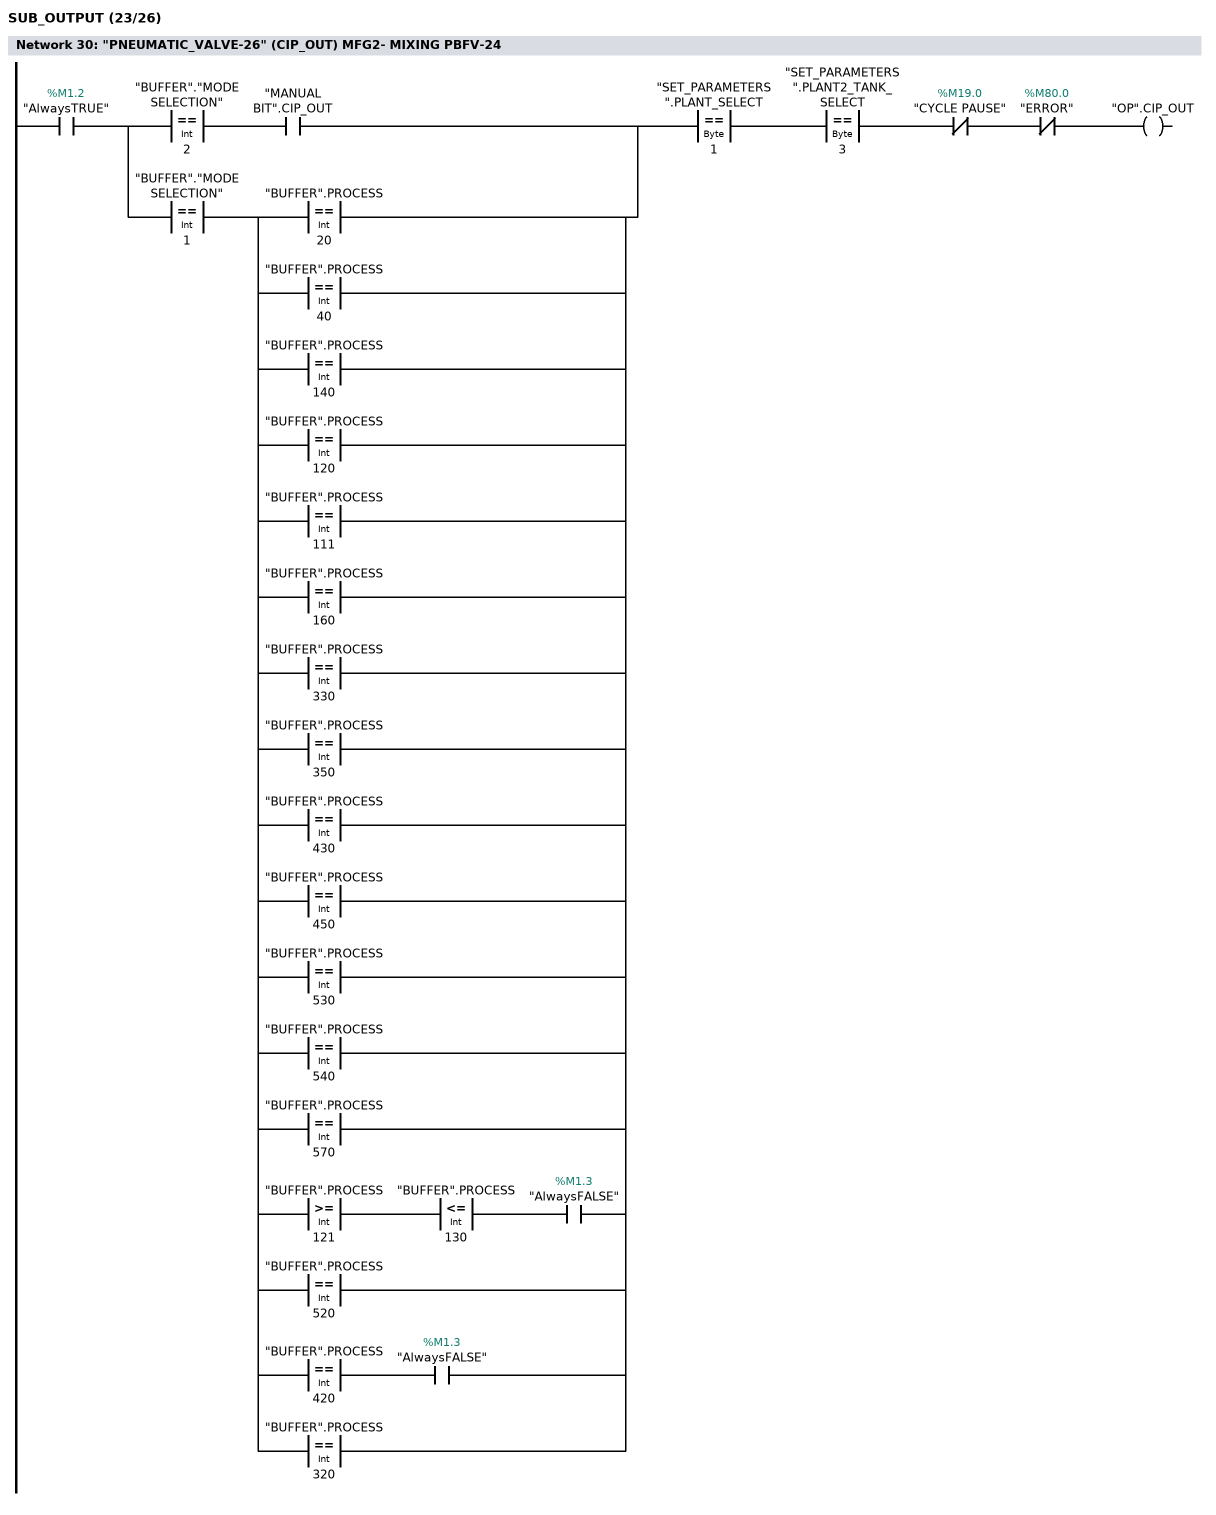
   RUNG wire#powerrail
      Contact( "AlwaysTRUE" )
      wire#w1
      { S7_Templates := "SrcType := Int" } EQ_Contact(in1 := "BUFFER"."MODE SELECTION", in2 := 2)
      Contact( "MANUAL BIT".CIP_OUT )
      wire#w2
      { S7_Templates := "SrcType := Byte" } EQ_Contact(in1 := "SET_PARAMETERS".PLANT_SELECT, in2 := 1)
      { S7_Templates := "SrcType := Byte" } EQ_Contact(in1 := "SET_PARAMETERS".PLANT2_TANK_SELECT, in2 := 3)
      I_Contact( "CYCLE PAUSE" )
      I_Contact( "ERROR" )
      Coil( "OP".CIP_OUT )
   END_RUNG
   RUNG wire#w1
      { S7_Templates := "SrcType := Int" } EQ_Contact(in1 := "BUFFER"."MODE SELECTION", in2 := 1)
      wire#w3
      { S7_Templates := "SrcType := Int" } EQ_Contact(in1 := "BUFFER".PROCESS, in2 := 20)
   END_RUNG wire#w2
   RUNG wire#w3
      { S7_Templates := "SrcType := Int" } EQ_Contact(in1 := "BUFFER".PROCESS, in2 := 40)
   END_RUNG wire#w2
   RUNG wire#w3
      { S7_Templates := "SrcType := Int" } EQ_Contact(in1 := "BUFFER".PROCESS, in2 := 140)
   END_RUNG wire#w2
   RUNG wire#w3
      { S7_Templates := "SrcType := Int" } EQ_Contact(in1 := "BUFFER".PROCESS, in2 := 120)
   END_RUNG wire#w2
   RUNG wire#w3
      { S7_Templates := "SrcType := Int" } EQ_Contact(in1 := "BUFFER".PROCESS, in2 := 111)
   END_RUNG wire#w2
   RUNG wire#w3
      { S7_Templates := "SrcType := Int" } EQ_Contact(in1 := "BUFFER".PROCESS, in2 := 160)
   END_RUNG wire#w2
   RUNG wire#w3
      { S7_Templates := "SrcType := Int" } EQ_Contact(in1 := "BUFFER".PROCESS, in2 := 330)
   END_RUNG wire#w2
   RUNG wire#w3
      { S7_Templates := "SrcType := Int" } EQ_Contact(in1 := "BUFFER".PROCESS, in2 := 350)
   END_RUNG wire#w2
   RUNG wire#w3
      { S7_Templates := "SrcType := Int" } EQ_Contact(in1 := "BUFFER".PROCESS, in2 := 430)
   END_RUNG wire#w2
   RUNG wire#w3
      { S7_Templates := "SrcType := Int" } EQ_Contact(in1 := "BUFFER".PROCESS, in2 := 450)
   END_RUNG wire#w2
   RUNG wire#w3
      { S7_Templates := "SrcType := Int" } EQ_Contact(in1 := "BUFFER".PROCESS, in2 := 530)
   END_RUNG wire#w2
   RUNG wire#w3
      { S7_Templates := "SrcType := Int" } EQ_Contact(in1 := "BUFFER".PROCESS, in2 := 540)
   END_RUNG wire#w2
   RUNG wire#w3
      { S7_Templates := "SrcType := Int" } EQ_Contact(in1 := "BUFFER".PROCESS, in2 := 570)
   END_RUNG wire#w2
   RUNG wire#w3
      { S7_Templates := "SrcType := Int" } GE_Contact(in1 := "BUFFER".PROCESS, in2 := 121)
      { S7_Templates := "SrcType := Int" } LE_Contact(in1 := "BUFFER".PROCESS, in2 := 130)
      Contact( "AlwaysFALSE" )
   END_RUNG wire#w2
   RUNG wire#w3
      { S7_Templates := "SrcType := Int" } EQ_Contact(in1 := "BUFFER".PROCESS, in2 := 520)
   END_RUNG wire#w2
   RUNG wire#w3
      { S7_Templates := "SrcType := Int" } EQ_Contact(in1 := "BUFFER".PROCESS, in2 := 420)
      Contact( "AlwaysFALSE" )
   END_RUNG wire#w2
   RUNG wire#w3
      { S7_Templates := "SrcType := Int" } EQ_Contact(in1 := "BUFFER".PROCESS, in2 := 320)
   END_RUNG wire#w2
   // the same network as SCL:
   "OP".CIP_OUT := "AlwaysTRUE" AND ((("BUFFER"."MODE SELECTION" = 2) AND "MANUAL BIT".CIP_OUT) OR (("BUFFER"."MODE SELECTION" = 1) AND (("BUFFER".PROCESS = 20) OR ("BUFFER".PROCESS = 40) OR ("BUFFER".PROCESS = 140) OR ("BUFFER".PROCESS = 120) OR ("BUFFER".PROCESS = 111) OR ("BUFFER".PROCESS = 160) OR ("BUFFER".PROCESS = 330) OR ("BUFFER".PROCESS = 350) OR ("BUFFER".PROCESS = 430) OR ("BUFFER".PROCESS = 450) OR ("BUFFER".PROCESS = 530) OR ("BUFFER".PROCESS = 540) OR ("BUFFER".PROCESS = 570) OR (("BUFFER".PROCESS >= 121) AND ("BUFFER".PROCESS <= 130) AND "AlwaysFALSE") OR ("BUFFER".PROCESS = 520) OR (("BUFFER".PROCESS = 420) AND "AlwaysFALSE") OR ("BUFFER".PROCESS = 320)))) AND ("SET_PARAMETERS".PLANT_SELECT = 1) AND ("SET_PARAMETERS".PLANT2_TANK_SELECT = 3) AND NOT "CYCLE PAUSE" AND NOT "ERROR";
END_REGION

REGION Network 32: reset 18 and 25
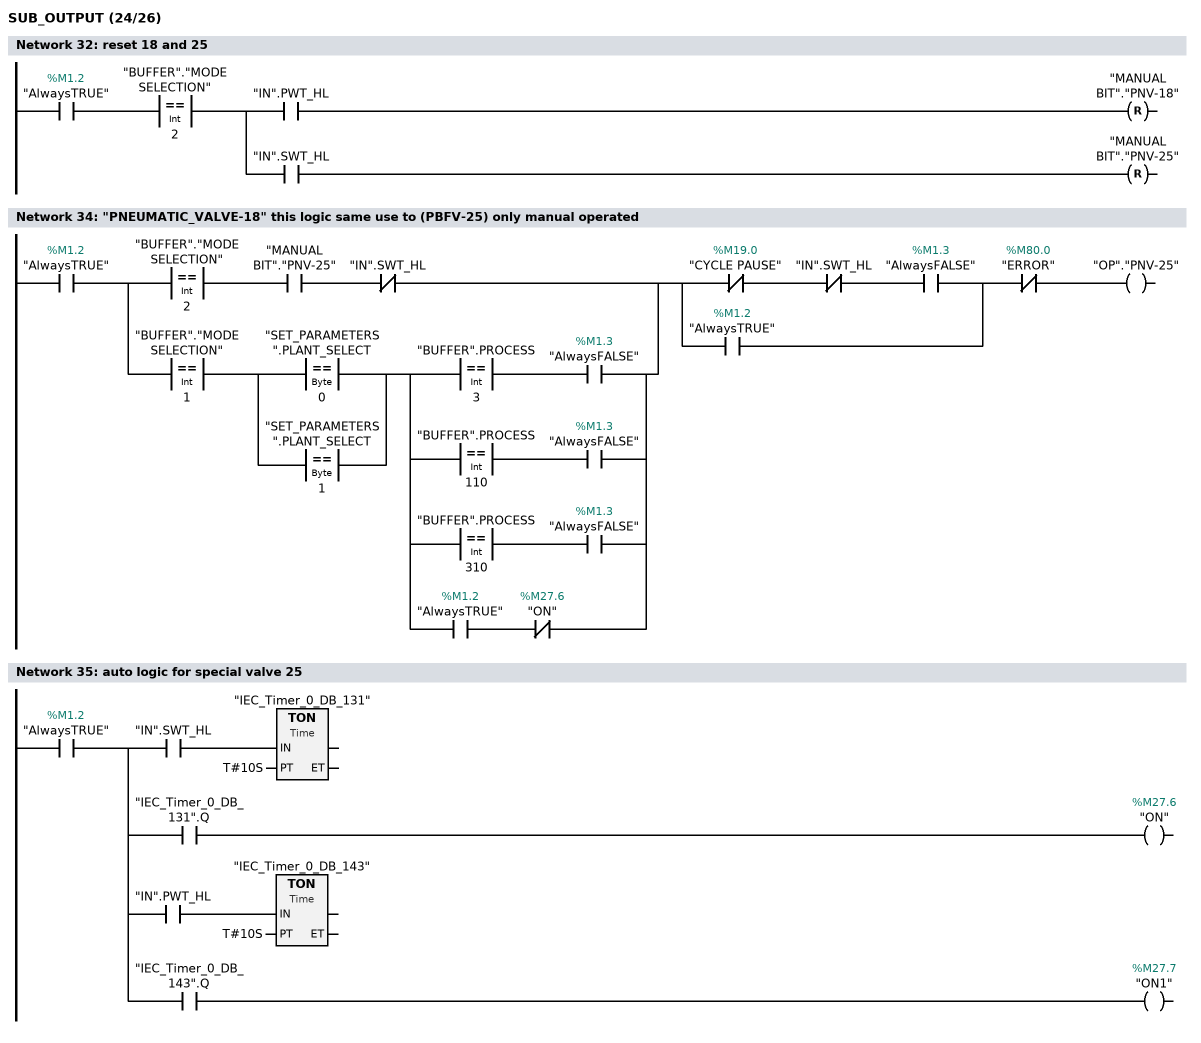
   RUNG wire#powerrail
      Contact( "AlwaysTRUE" )
      { S7_Templates := "SrcType := Int" } EQ_Contact(in1 := "BUFFER"."MODE SELECTION", in2 := 2)
      wire#w1
      Contact( "IN".PWT_HL )
      R_Coil( "MANUAL BIT"."PNV-18" )
   END_RUNG
   RUNG wire#w1
      Contact( "IN".SWT_HL )
      R_Coil( "MANUAL BIT"."PNV-25" )
   END_RUNG
   // the same network as SCL:
   #_w1 := "AlwaysTRUE" AND ("BUFFER"."MODE SELECTION" = 2);
   IF #_w1 AND "IN".PWT_HL THEN "MANUAL BIT"."PNV-18" := FALSE; END_IF;
   IF #_w1 AND "IN".SWT_HL THEN "MANUAL BIT"."PNV-25" := FALSE; END_IF;
END_REGION

REGION Network 34: "PNEUMATIC_VALVE-18" this logic same use to (PBFV-25) only manual operated
   RUNG wire#powerrail
      Contact( "AlwaysTRUE" )
      wire#w1
      { S7_Templates := "SrcType := Int" } EQ_Contact(in1 := "BUFFER"."MODE SELECTION", in2 := 2)
      Contact( "MANUAL BIT"."PNV-25" )
      I_Contact( "IN".SWT_HL )
      wire#w2
      I_Contact( "CYCLE PAUSE" )
      I_Contact( "IN".SWT_HL )
      Contact( "AlwaysFALSE" )
      wire#w5
      I_Contact( "ERROR" )
      Coil( "OP"."PNV-25" )
   END_RUNG
   RUNG wire#w1
      { S7_Templates := "SrcType := Int" } EQ_Contact(in1 := "BUFFER"."MODE SELECTION", in2 := 1)
      wire#w3
      { S7_Templates := "SrcType := Byte" } EQ_Contact(in1 := "SET_PARAMETERS".PLANT_SELECT, in2 := 0)
      wire#w4
      { S7_Templates := "SrcType := Int" } EQ_Contact(in1 := "BUFFER".PROCESS, in2 := 3)
      Contact( "AlwaysFALSE" )
   END_RUNG wire#w2
   RUNG wire#w3
      { S7_Templates := "SrcType := Byte" } EQ_Contact(in1 := "SET_PARAMETERS".PLANT_SELECT, in2 := 1)
   END_RUNG wire#w4
   RUNG wire#w4
      { S7_Templates := "SrcType := Int" } EQ_Contact(in1 := "BUFFER".PROCESS, in2 := 110)
      Contact( "AlwaysFALSE" )
   END_RUNG wire#w2
   RUNG wire#w4
      { S7_Templates := "SrcType := Int" } EQ_Contact(in1 := "BUFFER".PROCESS, in2 := 310)
      Contact( "AlwaysFALSE" )
   END_RUNG wire#w2
   RUNG wire#w4
      Contact( "AlwaysTRUE" )
      I_Contact( "ON" )
   END_RUNG wire#w2
   RUNG wire#w2
      Contact( "AlwaysTRUE" )
   END_RUNG wire#w5
   // the same network as SCL:
   "OP"."PNV-25" := "AlwaysTRUE" AND ((("BUFFER"."MODE SELECTION" = 2) AND "MANUAL BIT"."PNV-25" AND NOT "IN".SWT_HL) OR (("BUFFER"."MODE SELECTION" = 1) AND (("SET_PARAMETERS".PLANT_SELECT = 0) OR ("SET_PARAMETERS".PLANT_SELECT = 1)) AND ((("BUFFER".PROCESS = 3) AND "AlwaysFALSE") OR (("BUFFER".PROCESS = 110) AND "AlwaysFALSE") OR (("BUFFER".PROCESS = 310) AND "AlwaysFALSE") OR ("AlwaysTRUE" AND NOT "ON")))) AND ((NOT "CYCLE PAUSE" AND NOT "IN".SWT_HL AND "AlwaysFALSE") OR "AlwaysTRUE") AND NOT "ERROR";
END_REGION

REGION Network 35: auto logic for special valve 25
   RUNG wire#powerrail
      Contact( "AlwaysTRUE" )
      wire#w1
      Contact( "IN".SWT_HL )
      { S7_Templates := "time_type := Time" } "IEC_Timer_0_DB_131".TON(pt := T#10S, et =>)
   END_RUNG
   RUNG wire#w1
      Contact( "IEC_Timer_0_DB_131".Q )
      Coil( "ON" )
   END_RUNG
   RUNG wire#w1
      Contact( "IN".PWT_HL )
      { S7_Templates := "time_type := Time" } "IEC_Timer_0_DB_143".TON(pt := T#10S, et =>)
   END_RUNG
   RUNG wire#w1
      Contact( "IEC_Timer_0_DB_143".Q )
      Coil( "ON1" )
   END_RUNG
   // the same network as SCL:
   "IEC_Timer_0_DB_131".TON(IN := "AlwaysTRUE" AND "IN".SWT_HL, PT := T#10S);
   "ON" := "AlwaysTRUE" AND "IEC_Timer_0_DB_131".Q;
   "IEC_Timer_0_DB_143".TON(IN := "AlwaysTRUE" AND "IN".PWT_HL, PT := T#10S);
   "ON1" := "AlwaysTRUE" AND "IEC_Timer_0_DB_143".Q;
END_REGION

REGION Network 36: valve 22 time base final rinse 1 b type cycle
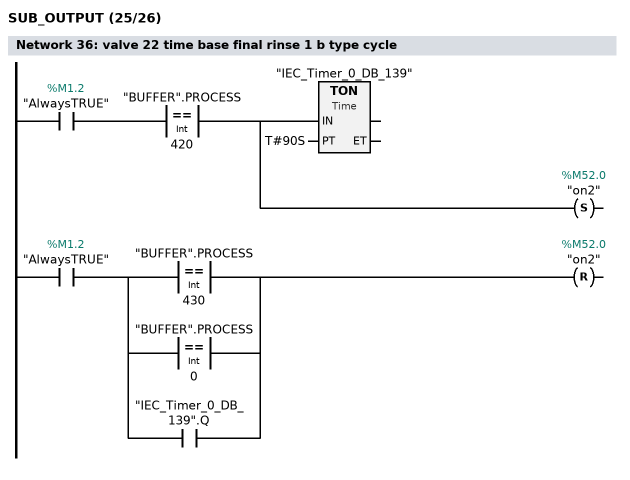
   RUNG wire#powerrail
      Contact( "AlwaysTRUE" )
      { S7_Templates := "SrcType := Int" } EQ_Contact(in1 := "BUFFER".PROCESS, in2 := 420)
      wire#w1
      { S7_Templates := "time_type := Time" } "IEC_Timer_0_DB_139".TON(pt := T#90S, et =>)
   END_RUNG
   RUNG wire#w1
      S_Coil( "on2" )
   END_RUNG
   RUNG wire#powerrail
      Contact( "AlwaysTRUE" )
      wire#w2
      { S7_Templates := "SrcType := Int" } EQ_Contact(in1 := "BUFFER".PROCESS, in2 := 430)
      wire#w3
      R_Coil( "on2" )
   END_RUNG
   RUNG wire#w2
      { S7_Templates := "SrcType := Int" } EQ_Contact(in1 := "BUFFER".PROCESS, in2 := 0)
   END_RUNG wire#w3
   RUNG wire#w2
      Contact( "IEC_Timer_0_DB_139".Q )
   END_RUNG wire#w3
   // the same network as SCL:
   #_w1 := "AlwaysTRUE" AND ("BUFFER".PROCESS = 420);
   "IEC_Timer_0_DB_139".TON(IN := #_w1, PT := T#90S);
   IF #_w1 THEN "on2" := TRUE; END_IF;
   IF "AlwaysTRUE" AND (("BUFFER".PROCESS = 430) OR ("BUFFER".PROCESS = 0) OR "IEC_Timer_0_DB_139".Q) THEN
       "on2" := FALSE;
   END_IF;
END_REGION

REGION Network 37: for air purpose will be on 5sec valve11
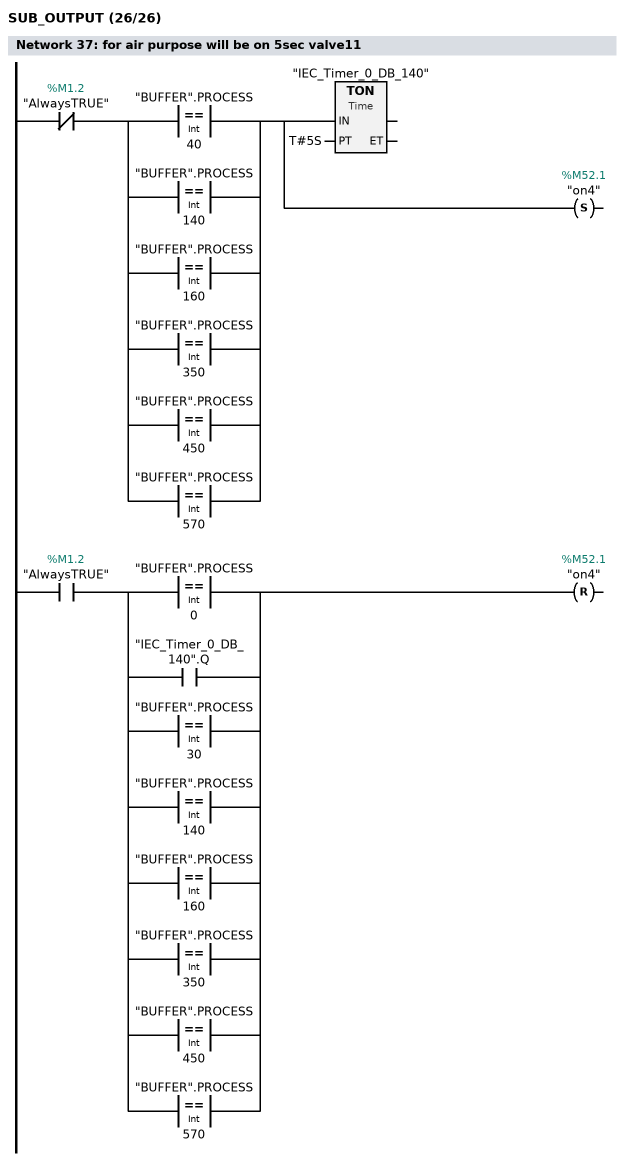
   RUNG wire#powerrail
      I_Contact( "AlwaysTRUE" )
      wire#w1
      { S7_Templates := "SrcType := Int" } EQ_Contact(in1 := "BUFFER".PROCESS, in2 := 40)
      wire#w2
      { S7_Templates := "time_type := Time" } "IEC_Timer_0_DB_140".TON(pt := T#5S, et =>)
   END_RUNG
   RUNG wire#w1
      { S7_Templates := "SrcType := Int" } EQ_Contact(in1 := "BUFFER".PROCESS, in2 := 140)
   END_RUNG wire#w2
   RUNG wire#w1
      { S7_Templates := "SrcType := Int" } EQ_Contact(in1 := "BUFFER".PROCESS, in2 := 160)
   END_RUNG wire#w2
   RUNG wire#w1
      { S7_Templates := "SrcType := Int" } EQ_Contact(in1 := "BUFFER".PROCESS, in2 := 350)
   END_RUNG wire#w2
   RUNG wire#w1
      { S7_Templates := "SrcType := Int" } EQ_Contact(in1 := "BUFFER".PROCESS, in2 := 450)
   END_RUNG wire#w2
   RUNG wire#w1
      { S7_Templates := "SrcType := Int" } EQ_Contact(in1 := "BUFFER".PROCESS, in2 := 570)
   END_RUNG wire#w2
   RUNG wire#w2
      S_Coil( "on4" )
   END_RUNG
   RUNG wire#powerrail
      Contact( "AlwaysTRUE" )
      wire#w3
      { S7_Templates := "SrcType := Int" } EQ_Contact(in1 := "BUFFER".PROCESS, in2 := 0)
      wire#w4
      R_Coil( "on4" )
   END_RUNG
   RUNG wire#w3
      Contact( "IEC_Timer_0_DB_140".Q )
   END_RUNG wire#w4
   RUNG wire#w3
      { S7_Templates := "SrcType := Int" } EQ_Contact(in1 := "BUFFER".PROCESS, in2 := 30)
   END_RUNG wire#w4
   RUNG wire#w3
      { S7_Templates := "SrcType := Int" } EQ_Contact(in1 := "BUFFER".PROCESS, in2 := 140)
   END_RUNG wire#w4
   RUNG wire#w3
      { S7_Templates := "SrcType := Int" } EQ_Contact(in1 := "BUFFER".PROCESS, in2 := 160)
   END_RUNG wire#w4
   RUNG wire#w3
      { S7_Templates := "SrcType := Int" } EQ_Contact(in1 := "BUFFER".PROCESS, in2 := 350)
   END_RUNG wire#w4
   RUNG wire#w3
      { S7_Templates := "SrcType := Int" } EQ_Contact(in1 := "BUFFER".PROCESS, in2 := 450)
   END_RUNG wire#w4
   RUNG wire#w3
      { S7_Templates := "SrcType := Int" } EQ_Contact(in1 := "BUFFER".PROCESS, in2 := 570)
   END_RUNG wire#w4
   // the same network as SCL:
   #_w1 := NOT "AlwaysTRUE" AND (("BUFFER".PROCESS = 40) OR ("BUFFER".PROCESS = 140) OR ("BUFFER".PROCESS = 160) OR ("BUFFER".PROCESS = 350) OR ("BUFFER".PROCESS = 450) OR ("BUFFER".PROCESS = 570));
   "IEC_Timer_0_DB_140".TON(IN := #_w1, PT := T#5S);
   IF #_w1 THEN "on4" := TRUE; END_IF;
   IF "AlwaysTRUE" AND (("BUFFER".PROCESS = 0) OR "IEC_Timer_0_DB_140".Q OR ("BUFFER".PROCESS = 30) OR ("BUFFER".PROCESS = 140) OR ("BUFFER".PROCESS = 160) OR ("BUFFER".PROCESS = 350) OR ("BUFFER".PROCESS = 450) OR ("BUFFER".PROCESS = 570)) THEN
       "on4" := FALSE;
   END_IF;
END_REGION
END_FUNCTION

FUNCTION "RECIPE" : Void   // FC7, LAD
{ S7_Optimized_Access := 'TRUE' }
// stored: SetENOAutomatically false
BEGIN

REGION Network 1: RINSE 1
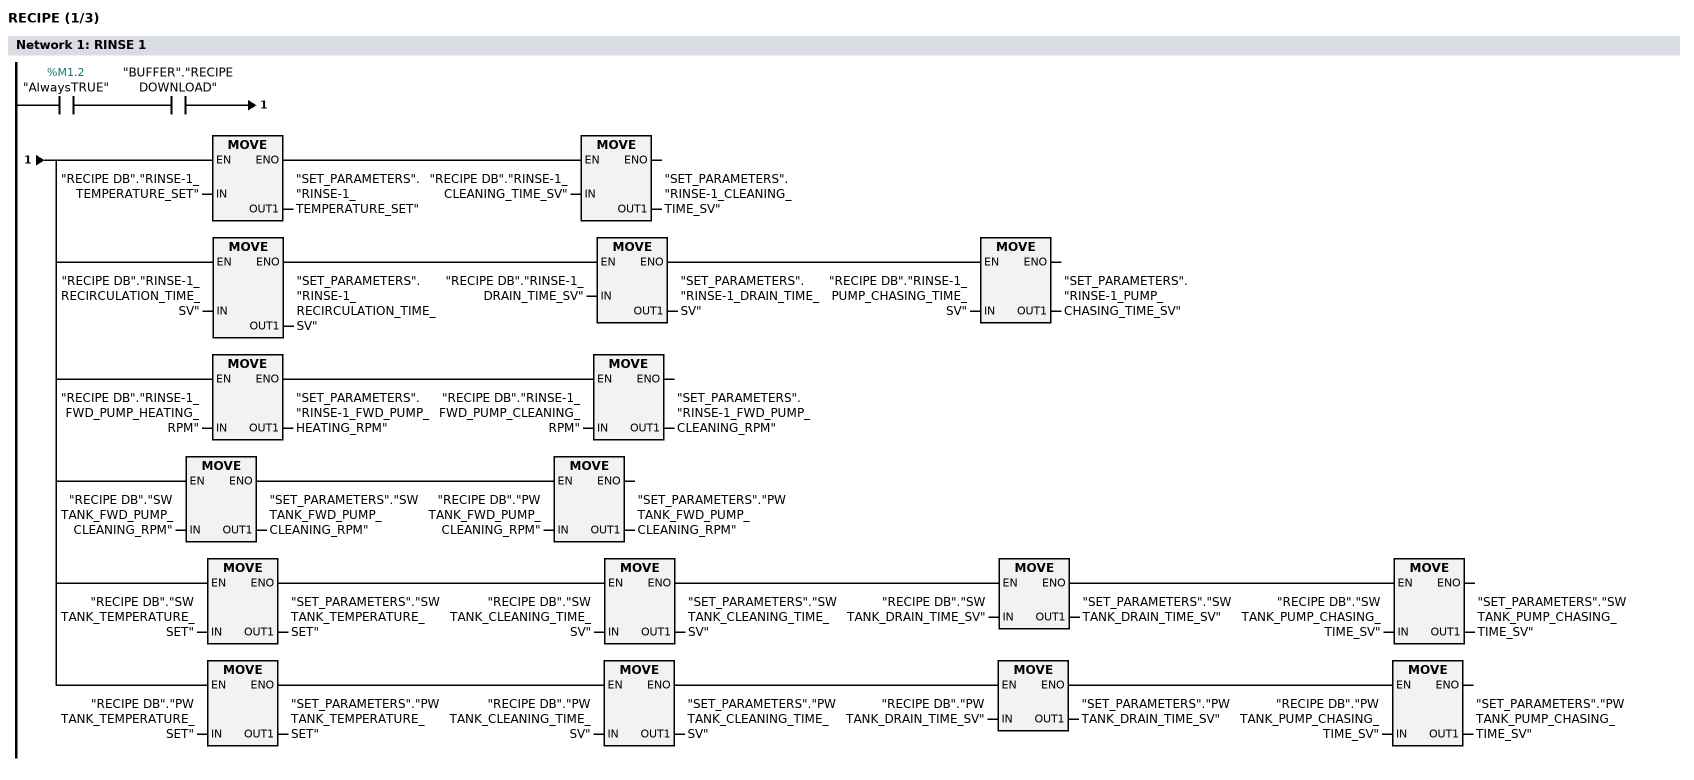
   RUNG wire#powerrail
      Contact( "AlwaysTRUE" )
      Contact( "BUFFER"."RECIPE DOWNLOAD" )
      wire#w1
      Move(in := "RECIPE DB"."RINSE-1_TEMPERATURE_SET", out1 => "SET_PARAMETERS"."RINSE-1_TEMPERATURE_SET")
      Move(in := "RECIPE DB"."RINSE-1_CLEANING_TIME_SV", out1 => "SET_PARAMETERS"."RINSE-1_CLEANING_TIME_SV")
   END_RUNG
   RUNG wire#w1
      Move(in := "RECIPE DB"."RINSE-1_RECIRCULATION_TIME_SV", out1 => "SET_PARAMETERS"."RINSE-1_RECIRCULATION_TIME_SV")
      Move(in := "RECIPE DB"."RINSE-1_DRAIN_TIME_SV", out1 => "SET_PARAMETERS"."RINSE-1_DRAIN_TIME_SV")
      Move(in := "RECIPE DB"."RINSE-1_PUMP_CHASING_TIME_SV", out1 => "SET_PARAMETERS"."RINSE-1_PUMP_CHASING_TIME_SV")
   END_RUNG
   RUNG wire#w1
      Move(in := "RECIPE DB"."RINSE-1_FWD_PUMP_HEATING_RPM", out1 => "SET_PARAMETERS"."RINSE-1_FWD_PUMP_HEATING_RPM")
      Move(in := "RECIPE DB"."RINSE-1_FWD_PUMP_CLEANING_RPM", out1 => "SET_PARAMETERS"."RINSE-1_FWD_PUMP_CLEANING_RPM")
   END_RUNG
   RUNG wire#w1
      Move(in := "RECIPE DB"."SW TANK_FWD_PUMP_CLEANING_RPM", out1 => "SET_PARAMETERS"."SW TANK_FWD_PUMP_CLEANING_RPM")
      Move(in := "RECIPE DB"."PW TANK_FWD_PUMP_CLEANING_RPM", out1 => "SET_PARAMETERS"."PW TANK_FWD_PUMP_CLEANING_RPM")
   END_RUNG
   RUNG wire#w1
      Move(in := "RECIPE DB"."SW TANK_TEMPERATURE_SET", out1 => "SET_PARAMETERS"."SW TANK_TEMPERATURE_SET")
      Move(in := "RECIPE DB"."SW TANK_CLEANING_TIME_SV", out1 => "SET_PARAMETERS"."SW TANK_CLEANING_TIME_SV")
      Move(in := "RECIPE DB"."SW TANK_DRAIN_TIME_SV", out1 => "SET_PARAMETERS"."SW TANK_DRAIN_TIME_SV")
      Move(in := "RECIPE DB"."SW TANK_PUMP_CHASING_TIME_SV", out1 => "SET_PARAMETERS"."SW TANK_PUMP_CHASING_TIME_SV")
   END_RUNG
   RUNG wire#w1
      Move(in := "RECIPE DB"."PW TANK_TEMPERATURE_SET", out1 => "SET_PARAMETERS"."PW TANK_TEMPERATURE_SET")
      Move(in := "RECIPE DB"."PW TANK_CLEANING_TIME_SV", out1 => "SET_PARAMETERS"."PW TANK_CLEANING_TIME_SV")
      Move(in := "RECIPE DB"."PW TANK_DRAIN_TIME_SV", out1 => "SET_PARAMETERS"."PW TANK_DRAIN_TIME_SV")
      Move(in := "RECIPE DB"."PW TANK_PUMP_CHASING_TIME_SV", out1 => "SET_PARAMETERS"."PW TANK_PUMP_CHASING_TIME_SV")
   END_RUNG
   // the same network as SCL:
   IF "AlwaysTRUE" AND "BUFFER"."RECIPE DOWNLOAD" THEN
       "SET_PARAMETERS"."RINSE-1_TEMPERATURE_SET" := "RECIPE DB"."RINSE-1_TEMPERATURE_SET";
       "SET_PARAMETERS"."RINSE-1_CLEANING_TIME_SV" := "RECIPE DB"."RINSE-1_CLEANING_TIME_SV";
       "SET_PARAMETERS"."RINSE-1_RECIRCULATION_TIME_SV" := "RECIPE DB"."RINSE-1_RECIRCULATION_TIME_SV";
       "SET_PARAMETERS"."RINSE-1_DRAIN_TIME_SV" := "RECIPE DB"."RINSE-1_DRAIN_TIME_SV";
       "SET_PARAMETERS"."RINSE-1_PUMP_CHASING_TIME_SV" := "RECIPE DB"."RINSE-1_PUMP_CHASING_TIME_SV";
       "SET_PARAMETERS"."RINSE-1_FWD_PUMP_HEATING_RPM" := "RECIPE DB"."RINSE-1_FWD_PUMP_HEATING_RPM";
       "SET_PARAMETERS"."RINSE-1_FWD_PUMP_CLEANING_RPM" := "RECIPE DB"."RINSE-1_FWD_PUMP_CLEANING_RPM";
       "SET_PARAMETERS"."SW TANK_FWD_PUMP_CLEANING_RPM" := "RECIPE DB"."SW TANK_FWD_PUMP_CLEANING_RPM";
       "SET_PARAMETERS"."PW TANK_FWD_PUMP_CLEANING_RPM" := "RECIPE DB"."PW TANK_FWD_PUMP_CLEANING_RPM";
       "SET_PARAMETERS"."SW TANK_TEMPERATURE_SET" := "RECIPE DB"."SW TANK_TEMPERATURE_SET";
       "SET_PARAMETERS"."SW TANK_CLEANING_TIME_SV" := "RECIPE DB"."SW TANK_CLEANING_TIME_SV";
       "SET_PARAMETERS"."SW TANK_DRAIN_TIME_SV" := "RECIPE DB"."SW TANK_DRAIN_TIME_SV";
       "SET_PARAMETERS"."SW TANK_PUMP_CHASING_TIME_SV" := "RECIPE DB"."SW TANK_PUMP_CHASING_TIME_SV";
       "SET_PARAMETERS"."PW TANK_TEMPERATURE_SET" := "RECIPE DB"."PW TANK_TEMPERATURE_SET";
       "SET_PARAMETERS"."PW TANK_CLEANING_TIME_SV" := "RECIPE DB"."PW TANK_CLEANING_TIME_SV";
       "SET_PARAMETERS"."PW TANK_DRAIN_TIME_SV" := "RECIPE DB"."PW TANK_DRAIN_TIME_SV";
       "SET_PARAMETERS"."PW TANK_PUMP_CHASING_TIME_SV" := "RECIPE DB"."PW TANK_PUMP_CHASING_TIME_SV";
   END_IF;
END_REGION

REGION Network 2: WASH BY ACID / ALKALI
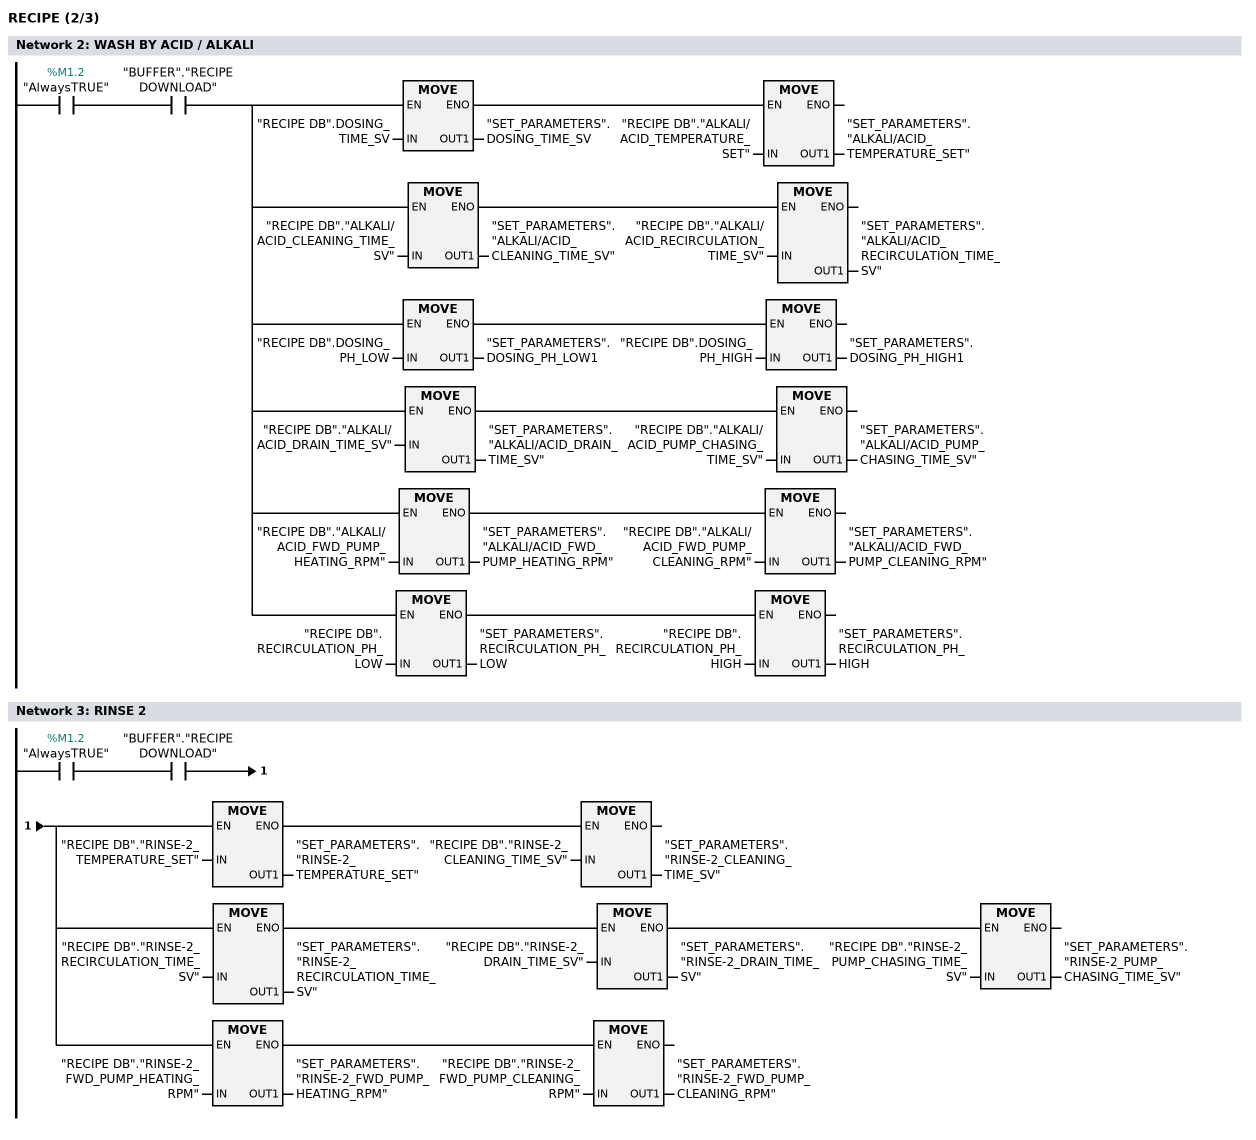
   RUNG wire#powerrail
      Contact( "AlwaysTRUE" )
      Contact( "BUFFER"."RECIPE DOWNLOAD" )
      wire#w1
      Move(in := "RECIPE DB".DOSING_TIME_SV, out1 => "SET_PARAMETERS".DOSING_TIME_SV)
      Move(in := "RECIPE DB"."ALKALI/ACID_TEMPERATURE_SET", out1 => "SET_PARAMETERS"."ALKALI/ACID_TEMPERATURE_SET")
   END_RUNG
   RUNG wire#w1
      Move(in := "RECIPE DB"."ALKALI/ACID_CLEANING_TIME_SV", out1 => "SET_PARAMETERS"."ALKALI/ACID_CLEANING_TIME_SV")
      Move(in := "RECIPE DB"."ALKALI/ACID_RECIRCULATION_TIME_SV", out1 => "SET_PARAMETERS"."ALKALI/ACID_RECIRCULATION_TIME_SV")
   END_RUNG
   RUNG wire#w1
      Move(in := "RECIPE DB".DOSING_PH_LOW, out1 => "SET_PARAMETERS".DOSING_PH_LOW1)
      Move(in := "RECIPE DB".DOSING_PH_HIGH, out1 => "SET_PARAMETERS".DOSING_PH_HIGH1)
   END_RUNG
   RUNG wire#w1
      Move(in := "RECIPE DB"."ALKALI/ACID_DRAIN_TIME_SV", out1 => "SET_PARAMETERS"."ALKALI/ACID_DRAIN_TIME_SV")
      Move(in := "RECIPE DB"."ALKALI/ACID_PUMP_CHASING_TIME_SV", out1 => "SET_PARAMETERS"."ALKALI/ACID_PUMP_CHASING_TIME_SV")
   END_RUNG
   RUNG wire#w1
      Move(in := "RECIPE DB"."ALKALI/ACID_FWD_PUMP_HEATING_RPM", out1 => "SET_PARAMETERS"."ALKALI/ACID_FWD_PUMP_HEATING_RPM")
      Move(in := "RECIPE DB"."ALKALI/ACID_FWD_PUMP_CLEANING_RPM", out1 => "SET_PARAMETERS"."ALKALI/ACID_FWD_PUMP_CLEANING_RPM")
   END_RUNG
   RUNG wire#w1
      Move(in := "RECIPE DB".RECIRCULATION_PH_LOW, out1 => "SET_PARAMETERS".RECIRCULATION_PH_LOW)
      Move(in := "RECIPE DB".RECIRCULATION_PH_HIGH, out1 => "SET_PARAMETERS".RECIRCULATION_PH_HIGH)
   END_RUNG
   // the same network as SCL:
   IF "AlwaysTRUE" AND "BUFFER"."RECIPE DOWNLOAD" THEN
       "SET_PARAMETERS".DOSING_TIME_SV := "RECIPE DB".DOSING_TIME_SV;
       "SET_PARAMETERS"."ALKALI/ACID_TEMPERATURE_SET" := "RECIPE DB"."ALKALI/ACID_TEMPERATURE_SET";
       "SET_PARAMETERS"."ALKALI/ACID_CLEANING_TIME_SV" := "RECIPE DB"."ALKALI/ACID_CLEANING_TIME_SV";
       "SET_PARAMETERS"."ALKALI/ACID_RECIRCULATION_TIME_SV" := "RECIPE DB"."ALKALI/ACID_RECIRCULATION_TIME_SV";
       "SET_PARAMETERS".DOSING_PH_LOW1 := "RECIPE DB".DOSING_PH_LOW;
       "SET_PARAMETERS".DOSING_PH_HIGH1 := "RECIPE DB".DOSING_PH_HIGH;
       "SET_PARAMETERS"."ALKALI/ACID_DRAIN_TIME_SV" := "RECIPE DB"."ALKALI/ACID_DRAIN_TIME_SV";
       "SET_PARAMETERS"."ALKALI/ACID_PUMP_CHASING_TIME_SV" := "RECIPE DB"."ALKALI/ACID_PUMP_CHASING_TIME_SV";
       "SET_PARAMETERS"."ALKALI/ACID_FWD_PUMP_HEATING_RPM" := "RECIPE DB"."ALKALI/ACID_FWD_PUMP_HEATING_RPM";
       "SET_PARAMETERS"."ALKALI/ACID_FWD_PUMP_CLEANING_RPM" := "RECIPE DB"."ALKALI/ACID_FWD_PUMP_CLEANING_RPM";
       "SET_PARAMETERS".RECIRCULATION_PH_LOW := "RECIPE DB".RECIRCULATION_PH_LOW;
       "SET_PARAMETERS".RECIRCULATION_PH_HIGH := "RECIPE DB".RECIRCULATION_PH_HIGH;
   END_IF;
END_REGION

REGION Network 3: RINSE 2
   RUNG wire#powerrail
      Contact( "AlwaysTRUE" )
      Contact( "BUFFER"."RECIPE DOWNLOAD" )
      wire#w1
      Move(in := "RECIPE DB"."RINSE-2_TEMPERATURE_SET", out1 => "SET_PARAMETERS"."RINSE-2_TEMPERATURE_SET")
      Move(in := "RECIPE DB"."RINSE-2_CLEANING_TIME_SV", out1 => "SET_PARAMETERS"."RINSE-2_CLEANING_TIME_SV")
   END_RUNG
   RUNG wire#w1
      Move(in := "RECIPE DB"."RINSE-2_RECIRCULATION_TIME_SV", out1 => "SET_PARAMETERS"."RINSE-2_RECIRCULATION_TIME_SV")
      Move(in := "RECIPE DB"."RINSE-2_DRAIN_TIME_SV", out1 => "SET_PARAMETERS"."RINSE-2_DRAIN_TIME_SV")
      Move(in := "RECIPE DB"."RINSE-2_PUMP_CHASING_TIME_SV", out1 => "SET_PARAMETERS"."RINSE-2_PUMP_CHASING_TIME_SV")
   END_RUNG
   RUNG wire#w1
      Move(in := "RECIPE DB"."RINSE-2_FWD_PUMP_HEATING_RPM", out1 => "SET_PARAMETERS"."RINSE-2_FWD_PUMP_HEATING_RPM")
      Move(in := "RECIPE DB"."RINSE-2_FWD_PUMP_CLEANING_RPM", out1 => "SET_PARAMETERS"."RINSE-2_FWD_PUMP_CLEANING_RPM")
   END_RUNG
   // the same network as SCL:
   IF "AlwaysTRUE" AND "BUFFER"."RECIPE DOWNLOAD" THEN
       "SET_PARAMETERS"."RINSE-2_TEMPERATURE_SET" := "RECIPE DB"."RINSE-2_TEMPERATURE_SET";
       "SET_PARAMETERS"."RINSE-2_CLEANING_TIME_SV" := "RECIPE DB"."RINSE-2_CLEANING_TIME_SV";
       "SET_PARAMETERS"."RINSE-2_RECIRCULATION_TIME_SV" := "RECIPE DB"."RINSE-2_RECIRCULATION_TIME_SV";
       "SET_PARAMETERS"."RINSE-2_DRAIN_TIME_SV" := "RECIPE DB"."RINSE-2_DRAIN_TIME_SV";
       "SET_PARAMETERS"."RINSE-2_PUMP_CHASING_TIME_SV" := "RECIPE DB"."RINSE-2_PUMP_CHASING_TIME_SV";
       "SET_PARAMETERS"."RINSE-2_FWD_PUMP_HEATING_RPM" := "RECIPE DB"."RINSE-2_FWD_PUMP_HEATING_RPM";
       "SET_PARAMETERS"."RINSE-2_FWD_PUMP_CLEANING_RPM" := "RECIPE DB"."RINSE-2_FWD_PUMP_CLEANING_RPM";
   END_IF;
END_REGION

REGION Network 4: RINSE 3 (FIANL_RINSE-1)
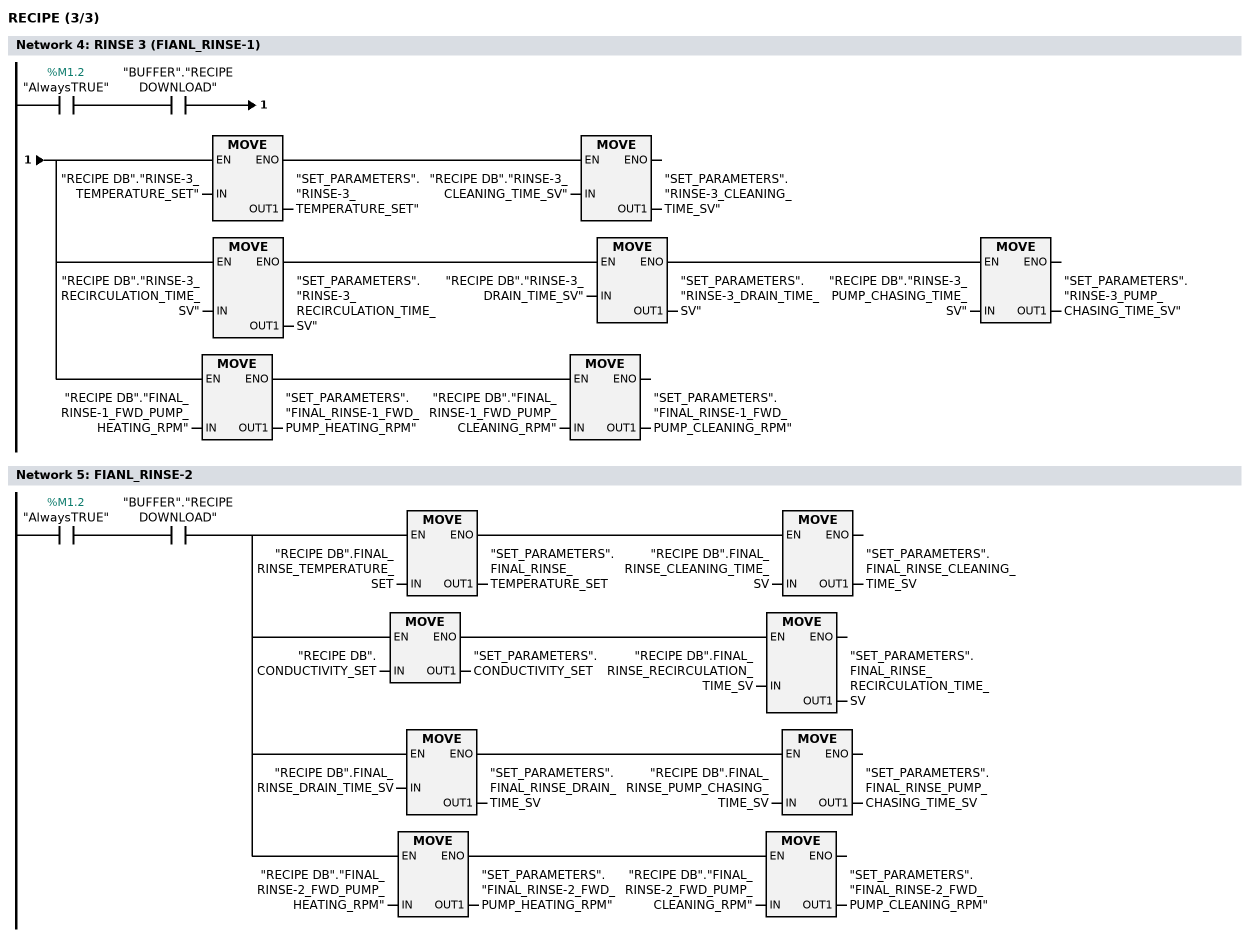
   RUNG wire#powerrail
      Contact( "AlwaysTRUE" )
      Contact( "BUFFER"."RECIPE DOWNLOAD" )
      wire#w1
      Move(in := "RECIPE DB"."RINSE-3_TEMPERATURE_SET", out1 => "SET_PARAMETERS"."RINSE-3_TEMPERATURE_SET")
      Move(in := "RECIPE DB"."RINSE-3_CLEANING_TIME_SV", out1 => "SET_PARAMETERS"."RINSE-3_CLEANING_TIME_SV")
   END_RUNG
   RUNG wire#w1
      Move(in := "RECIPE DB"."RINSE-3_RECIRCULATION_TIME_SV", out1 => "SET_PARAMETERS"."RINSE-3_RECIRCULATION_TIME_SV")
      Move(in := "RECIPE DB"."RINSE-3_DRAIN_TIME_SV", out1 => "SET_PARAMETERS"."RINSE-3_DRAIN_TIME_SV")
      Move(in := "RECIPE DB"."RINSE-3_PUMP_CHASING_TIME_SV", out1 => "SET_PARAMETERS"."RINSE-3_PUMP_CHASING_TIME_SV")
   END_RUNG
   RUNG wire#w1
      Move(in := "RECIPE DB"."FINAL_RINSE-1_FWD_PUMP_HEATING_RPM", out1 => "SET_PARAMETERS"."FINAL_RINSE-1_FWD_PUMP_HEATING_RPM")
      Move(in := "RECIPE DB"."FINAL_RINSE-1_FWD_PUMP_CLEANING_RPM", out1 => "SET_PARAMETERS"."FINAL_RINSE-1_FWD_PUMP_CLEANING_RPM")
   END_RUNG
   // the same network as SCL:
   IF "AlwaysTRUE" AND "BUFFER"."RECIPE DOWNLOAD" THEN
       "SET_PARAMETERS"."RINSE-3_TEMPERATURE_SET" := "RECIPE DB"."RINSE-3_TEMPERATURE_SET";
       "SET_PARAMETERS"."RINSE-3_CLEANING_TIME_SV" := "RECIPE DB"."RINSE-3_CLEANING_TIME_SV";
       "SET_PARAMETERS"."RINSE-3_RECIRCULATION_TIME_SV" := "RECIPE DB"."RINSE-3_RECIRCULATION_TIME_SV";
       "SET_PARAMETERS"."RINSE-3_DRAIN_TIME_SV" := "RECIPE DB"."RINSE-3_DRAIN_TIME_SV";
       "SET_PARAMETERS"."RINSE-3_PUMP_CHASING_TIME_SV" := "RECIPE DB"."RINSE-3_PUMP_CHASING_TIME_SV";
       "SET_PARAMETERS"."FINAL_RINSE-1_FWD_PUMP_HEATING_RPM" := "RECIPE DB"."FINAL_RINSE-1_FWD_PUMP_HEATING_RPM";
       "SET_PARAMETERS"."FINAL_RINSE-1_FWD_PUMP_CLEANING_RPM" := "RECIPE DB"."FINAL_RINSE-1_FWD_PUMP_CLEANING_RPM";
   END_IF;
END_REGION

REGION Network 5: FIANL_RINSE-2
   RUNG wire#powerrail
      Contact( "AlwaysTRUE" )
      Contact( "BUFFER"."RECIPE DOWNLOAD" )
      wire#w1
      Move(in := "RECIPE DB".FINAL_RINSE_TEMPERATURE_SET, out1 => "SET_PARAMETERS".FINAL_RINSE_TEMPERATURE_SET)
      Move(in := "RECIPE DB".FINAL_RINSE_CLEANING_TIME_SV, out1 => "SET_PARAMETERS".FINAL_RINSE_CLEANING_TIME_SV)
   END_RUNG
   RUNG wire#w1
      Move(in := "RECIPE DB".CONDUCTIVITY_SET, out1 => "SET_PARAMETERS".CONDUCTIVITY_SET)
      Move(in := "RECIPE DB".FINAL_RINSE_RECIRCULATION_TIME_SV, out1 => "SET_PARAMETERS".FINAL_RINSE_RECIRCULATION_TIME_SV)
   END_RUNG
   RUNG wire#w1
      Move(in := "RECIPE DB".FINAL_RINSE_DRAIN_TIME_SV, out1 => "SET_PARAMETERS".FINAL_RINSE_DRAIN_TIME_SV)
      Move(in := "RECIPE DB".FINAL_RINSE_PUMP_CHASING_TIME_SV, out1 => "SET_PARAMETERS".FINAL_RINSE_PUMP_CHASING_TIME_SV)
   END_RUNG
   RUNG wire#w1
      Move(in := "RECIPE DB"."FINAL_RINSE-2_FWD_PUMP_HEATING_RPM", out1 => "SET_PARAMETERS"."FINAL_RINSE-2_FWD_PUMP_HEATING_RPM")
      Move(in := "RECIPE DB"."FINAL_RINSE-2_FWD_PUMP_CLEANING_RPM", out1 => "SET_PARAMETERS"."FINAL_RINSE-2_FWD_PUMP_CLEANING_RPM")
   END_RUNG
   // the same network as SCL:
   IF "AlwaysTRUE" AND "BUFFER"."RECIPE DOWNLOAD" THEN
       "SET_PARAMETERS".FINAL_RINSE_TEMPERATURE_SET := "RECIPE DB".FINAL_RINSE_TEMPERATURE_SET;
       "SET_PARAMETERS".FINAL_RINSE_CLEANING_TIME_SV := "RECIPE DB".FINAL_RINSE_CLEANING_TIME_SV;
       "SET_PARAMETERS".CONDUCTIVITY_SET := "RECIPE DB".CONDUCTIVITY_SET;
       "SET_PARAMETERS".FINAL_RINSE_RECIRCULATION_TIME_SV := "RECIPE DB".FINAL_RINSE_RECIRCULATION_TIME_SV;
       "SET_PARAMETERS".FINAL_RINSE_DRAIN_TIME_SV := "RECIPE DB".FINAL_RINSE_DRAIN_TIME_SV;
       "SET_PARAMETERS".FINAL_RINSE_PUMP_CHASING_TIME_SV := "RECIPE DB".FINAL_RINSE_PUMP_CHASING_TIME_SV;
       "SET_PARAMETERS"."FINAL_RINSE-2_FWD_PUMP_HEATING_RPM" := "RECIPE DB"."FINAL_RINSE-2_FWD_PUMP_HEATING_RPM";
       "SET_PARAMETERS"."FINAL_RINSE-2_FWD_PUMP_CLEANING_RPM" := "RECIPE DB"."FINAL_RINSE-2_FWD_PUMP_CLEANING_RPM";
   END_IF;
END_REGION
END_FUNCTION

FUNCTION "DATE& TIME" : Void   // FC8, LAD
{ S7_Optimized_Access := 'TRUE' }
// stored: SetENOAutomatically false
BEGIN

REGION Network 1
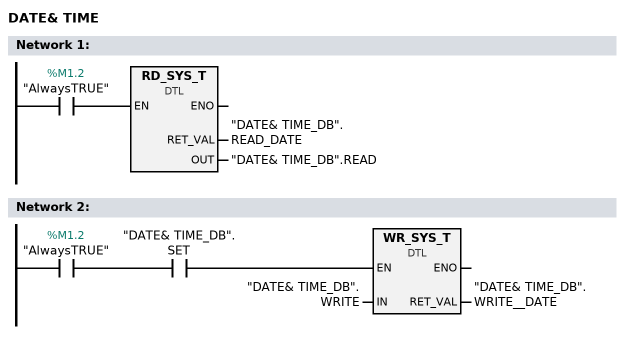
   RUNG wire#powerrail
      Contact( "AlwaysTRUE" )
      { S7_Templates := "date_type := DTL" } RD_SYS_T(RET_VAL => "DATE& TIME_DB".READ_DATE, OUT => "DATE& TIME_DB".READ)
   END_RUNG
   // the same network as SCL:
   IF "AlwaysTRUE" THEN "DATE& TIME_DB".READ_DATE := RD_SYS_T(OUT => "DATE& TIME_DB".READ); END_IF;
END_REGION

REGION Network 2
   RUNG wire#powerrail
      Contact( "AlwaysTRUE" )
      Contact( "DATE& TIME_DB".SET )
      { S7_Templates := "date_type := DTL" } WR_SYS_T(IN := "DATE& TIME_DB".WRITE, RET_VAL => "DATE& TIME_DB".WRITE__DATE)
   END_RUNG
   // the same network as SCL:
   IF "AlwaysTRUE" AND "DATE& TIME_DB".SET THEN
       "DATE& TIME_DB".WRITE__DATE := WR_SYS_T(IN := "DATE& TIME_DB".WRITE);
   END_IF;
END_REGION
END_FUNCTION

FUNCTION "ALARMS" : Void   // FC10, LAD
{ S7_Optimized_Access := 'TRUE' }
// stored: SetENOAutomatically false
   VAR_TEMP   // added for the SCL form of the ladder/FBD networks
      _w1 : Bool;
   END_VAR
BEGIN

REGION Network 1: ERROR BIT
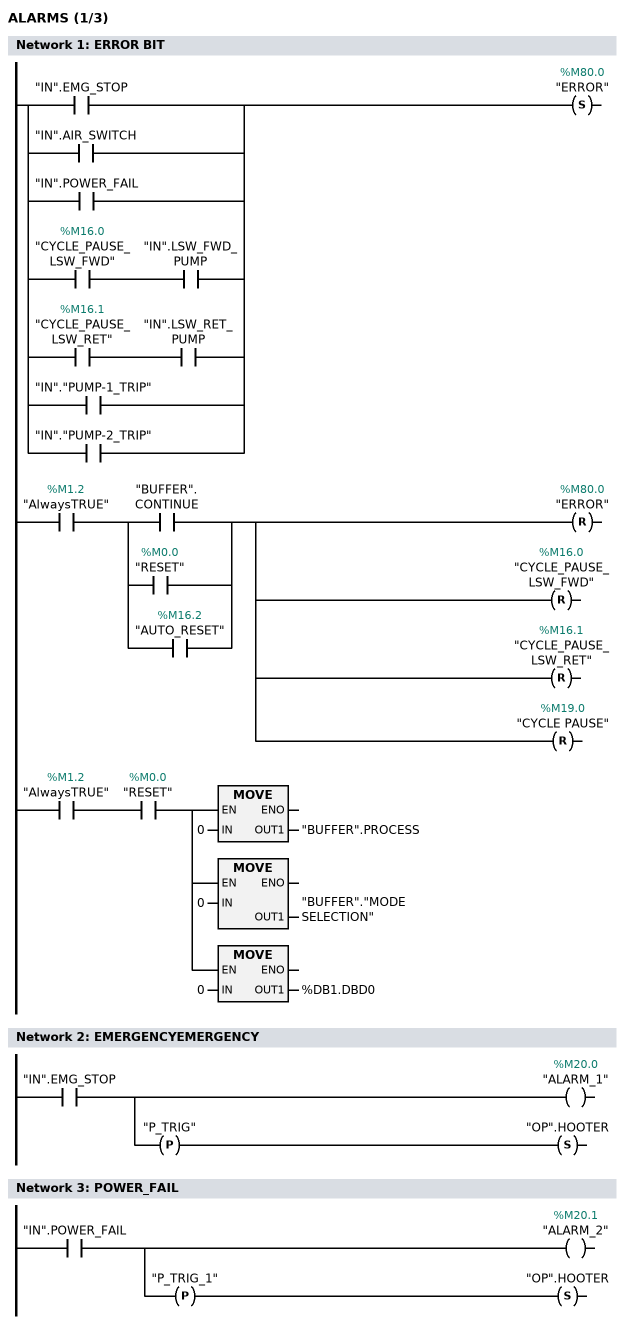
   RUNG wire#powerrail
      Contact( "IN".EMG_STOP )
      wire#w1
      S_Coil( "ERROR" )
   END_RUNG
   RUNG wire#powerrail
      Contact( "IN".AIR_SWITCH )
   END_RUNG wire#w1
   RUNG wire#powerrail
      Contact( "IN".POWER_FAIL )
   END_RUNG wire#w1
   RUNG wire#powerrail
      Contact( "CYCLE_PAUSE_LSW_FWD" )
      Contact( "IN".LSW_FWD_PUMP )
   END_RUNG wire#w1
   RUNG wire#powerrail
      Contact( "CYCLE_PAUSE_LSW_RET" )
      Contact( "IN".LSW_RET_PUMP )
   END_RUNG wire#w1
   RUNG wire#powerrail
      Contact( "IN"."PUMP-1_TRIP" )
   END_RUNG wire#w1
   RUNG wire#powerrail
      Contact( "IN"."PUMP-2_TRIP" )
   END_RUNG wire#w1
   RUNG wire#powerrail
      Contact( "AlwaysTRUE" )
      wire#w2
      Contact( "BUFFER".CONTINUE )
      wire#w3
      R_Coil( "ERROR" )
   END_RUNG
   RUNG wire#w2
      Contact( "RESET" )
   END_RUNG wire#w3
   RUNG wire#w2
      Contact( "AUTO_RESET" )
   END_RUNG wire#w3
   RUNG wire#w3
      R_Coil( "CYCLE_PAUSE_LSW_FWD" )
   END_RUNG
   RUNG wire#w3
      R_Coil( "CYCLE_PAUSE_LSW_RET" )
   END_RUNG
   RUNG wire#w3
      R_Coil( "CYCLE PAUSE" )
   END_RUNG
   RUNG wire#powerrail
      Contact( "AlwaysTRUE" )
      Contact( "RESET" )
      wire#w4
      Move(in := 0, out1 => "BUFFER".PROCESS)
   END_RUNG
   RUNG wire#w4
      Move(in := 0, out1 => "BUFFER"."MODE SELECTION")
   END_RUNG
   RUNG wire#w4
      Move(in := 0, out1 => %DB1.DBD0)
   END_RUNG
   // the same network as SCL:
   IF "IN".EMG_STOP OR "IN".AIR_SWITCH OR "IN".POWER_FAIL OR ("CYCLE_PAUSE_LSW_FWD" AND "IN".LSW_FWD_PUMP) OR ("CYCLE_PAUSE_LSW_RET" AND "IN".LSW_RET_PUMP) OR "IN"."PUMP-1_TRIP" OR "IN"."PUMP-2_TRIP" THEN
       "ERROR" := TRUE;
   END_IF;
   IF "AlwaysTRUE" AND ("BUFFER".CONTINUE OR "RESET" OR "AUTO_RESET") THEN
       "ERROR" := FALSE;
       "CYCLE_PAUSE_LSW_FWD" := FALSE;
       "CYCLE_PAUSE_LSW_RET" := FALSE;
       "CYCLE PAUSE" := FALSE;
   END_IF;
   IF "AlwaysTRUE" AND "RESET" THEN
       "BUFFER".PROCESS := 0;
       "BUFFER"."MODE SELECTION" := 0;
       %DB1.DBD0 := 0;
   END_IF;
END_REGION

REGION Network 2: EMERGENCYEMERGENCY
   RUNG wire#powerrail
      Contact( "IN".EMG_STOP )
      wire#w1
      Coil( "ALARM_1" )
   END_RUNG
   RUNG wire#w1
      P_Trig( "P_TRIG" )
      S_Coil( "OP".HOOTER )
   END_RUNG
   // the same network as SCL:
   "ALARM_1" := "IN".EMG_STOP;
   #_w1 := "IN".EMG_STOP AND NOT "P_TRIG";   // rising edge
   "P_TRIG" := "IN".EMG_STOP;
   IF #_w1 THEN "OP".HOOTER := TRUE; END_IF;
END_REGION

REGION Network 3: POWER_FAIL
   RUNG wire#powerrail
      Contact( "IN".POWER_FAIL )
      wire#w1
      Coil( "ALARM_2" )
   END_RUNG
   RUNG wire#w1
      P_Trig( "P_TRIG_1" )
      S_Coil( "OP".HOOTER )
   END_RUNG
   // the same network as SCL:
   "ALARM_2" := "IN".POWER_FAIL;
   #_w1 := "IN".POWER_FAIL AND NOT "P_TRIG_1";   // rising edge
   "P_TRIG_1" := "IN".POWER_FAIL;
   IF #_w1 THEN "OP".HOOTER := TRUE; END_IF;
END_REGION

REGION Network 4: FORWARD_PUMP_TRIP
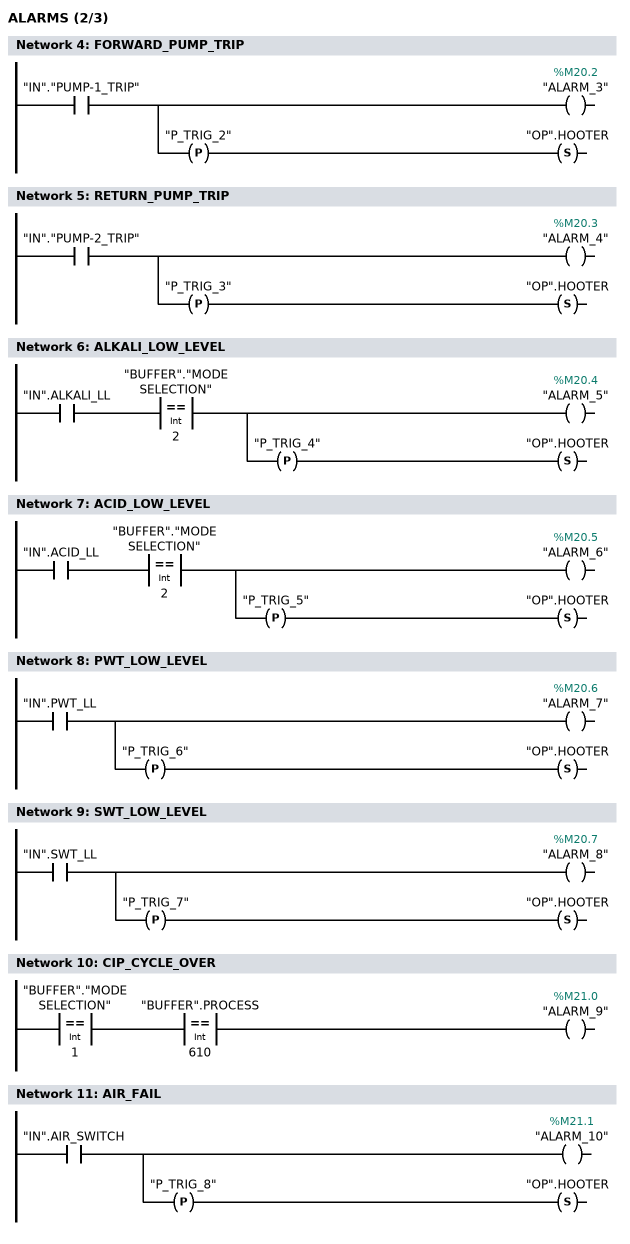
   RUNG wire#powerrail
      Contact( "IN"."PUMP-1_TRIP" )
      wire#w1
      Coil( "ALARM_3" )
   END_RUNG
   RUNG wire#w1
      P_Trig( "P_TRIG_2" )
      S_Coil( "OP".HOOTER )
   END_RUNG
   // the same network as SCL:
   "ALARM_3" := "IN"."PUMP-1_TRIP";
   #_w1 := "IN"."PUMP-1_TRIP" AND NOT "P_TRIG_2";   // rising edge
   "P_TRIG_2" := "IN"."PUMP-1_TRIP";
   IF #_w1 THEN "OP".HOOTER := TRUE; END_IF;
END_REGION

REGION Network 5: RETURN_PUMP_TRIP
   RUNG wire#powerrail
      Contact( "IN"."PUMP-2_TRIP" )
      wire#w1
      Coil( "ALARM_4" )
   END_RUNG
   RUNG wire#w1
      P_Trig( "P_TRIG_3" )
      S_Coil( "OP".HOOTER )
   END_RUNG
   // the same network as SCL:
   "ALARM_4" := "IN"."PUMP-2_TRIP";
   #_w1 := "IN"."PUMP-2_TRIP" AND NOT "P_TRIG_3";   // rising edge
   "P_TRIG_3" := "IN"."PUMP-2_TRIP";
   IF #_w1 THEN "OP".HOOTER := TRUE; END_IF;
END_REGION

REGION Network 6: ALKALI_LOW_LEVEL
   RUNG wire#powerrail
      Contact( "IN".ALKALI_LL )
      { S7_Templates := "SrcType := Int" } EQ_Contact(in1 := "BUFFER"."MODE SELECTION", in2 := 2)
      wire#w1
      Coil( "ALARM_5" )
   END_RUNG
   RUNG wire#w1
      P_Trig( "P_TRIG_4" )
      S_Coil( "OP".HOOTER )
   END_RUNG
   // the same network as SCL:
   "ALARM_5" := "IN".ALKALI_LL AND ("BUFFER"."MODE SELECTION" = 2);
   #_w1 := "ALARM_5" AND NOT "P_TRIG_4";   // rising edge
   "P_TRIG_4" := "ALARM_5";
   IF #_w1 THEN "OP".HOOTER := TRUE; END_IF;
END_REGION

REGION Network 7: ACID_LOW_LEVEL
   RUNG wire#powerrail
      Contact( "IN".ACID_LL )
      { S7_Templates := "SrcType := Int" } EQ_Contact(in1 := "BUFFER"."MODE SELECTION", in2 := 2)
      wire#w1
      Coil( "ALARM_6" )
   END_RUNG
   RUNG wire#w1
      P_Trig( "P_TRIG_5" )
      S_Coil( "OP".HOOTER )
   END_RUNG
   // the same network as SCL:
   "ALARM_6" := "IN".ACID_LL AND ("BUFFER"."MODE SELECTION" = 2);
   #_w1 := "ALARM_6" AND NOT "P_TRIG_5";   // rising edge
   "P_TRIG_5" := "ALARM_6";
   IF #_w1 THEN "OP".HOOTER := TRUE; END_IF;
END_REGION

REGION Network 8: PWT_LOW_LEVEL
   RUNG wire#powerrail
      Contact( "IN".PWT_LL )
      wire#w1
      Coil( "ALARM_7" )
   END_RUNG
   RUNG wire#w1
      P_Trig( "P_TRIG_6" )
      S_Coil( "OP".HOOTER )
   END_RUNG
   // the same network as SCL:
   "ALARM_7" := "IN".PWT_LL;
   #_w1 := "IN".PWT_LL AND NOT "P_TRIG_6";   // rising edge
   "P_TRIG_6" := "IN".PWT_LL;
   IF #_w1 THEN "OP".HOOTER := TRUE; END_IF;
END_REGION

REGION Network 9: SWT_LOW_LEVEL
   RUNG wire#powerrail
      Contact( "IN".SWT_LL )
      wire#w1
      Coil( "ALARM_8" )
   END_RUNG
   RUNG wire#w1
      P_Trig( "P_TRIG_7" )
      S_Coil( "OP".HOOTER )
   END_RUNG
   // the same network as SCL:
   "ALARM_8" := "IN".SWT_LL;
   #_w1 := "IN".SWT_LL AND NOT "P_TRIG_7";   // rising edge
   "P_TRIG_7" := "IN".SWT_LL;
   IF #_w1 THEN "OP".HOOTER := TRUE; END_IF;
END_REGION

REGION Network 10: CIP_CYCLE_OVER
   RUNG wire#powerrail
      { S7_Templates := "SrcType := Int" } EQ_Contact(in1 := "BUFFER"."MODE SELECTION", in2 := 1)
      { S7_Templates := "SrcType := Int" } EQ_Contact(in1 := "BUFFER".PROCESS, in2 := 610)
      Coil( "ALARM_9" )
   END_RUNG
   // the same network as SCL:
   "ALARM_9" := ("BUFFER"."MODE SELECTION" = 1) AND ("BUFFER".PROCESS = 610);
END_REGION

REGION Network 11: AIR_FAIL
   RUNG wire#powerrail
      Contact( "IN".AIR_SWITCH )
      wire#w1
      Coil( "ALARM_10" )
   END_RUNG
   RUNG wire#w1
      P_Trig( "P_TRIG_8" )
      S_Coil( "OP".HOOTER )
   END_RUNG
   // the same network as SCL:
   "ALARM_10" := "IN".AIR_SWITCH;
   #_w1 := "IN".AIR_SWITCH AND NOT "P_TRIG_8";   // rising edge
   "P_TRIG_8" := "IN".AIR_SWITCH;
   IF #_w1 THEN "OP".HOOTER := TRUE; END_IF;
END_REGION

REGION Network 12: FWD LSW_UNHEATHY_POPUP
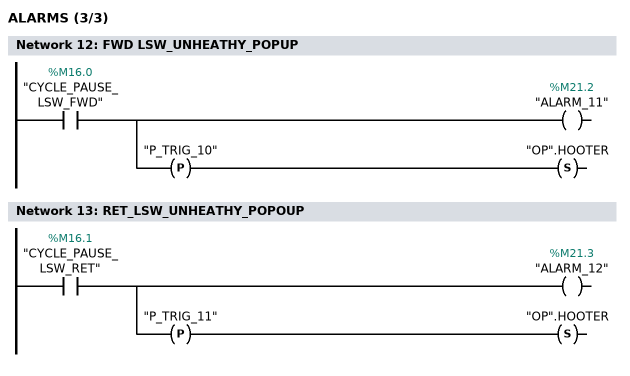
   RUNG wire#powerrail
      Contact( "CYCLE_PAUSE_LSW_FWD" )
      wire#w1
      Coil( "ALARM_11" )
   END_RUNG
   RUNG wire#w1
      P_Trig( "P_TRIG_10" )
      S_Coil( "OP".HOOTER )
   END_RUNG
   // the same network as SCL:
   "ALARM_11" := "CYCLE_PAUSE_LSW_FWD";
   #_w1 := "CYCLE_PAUSE_LSW_FWD" AND NOT "P_TRIG_10";   // rising edge
   "P_TRIG_10" := "CYCLE_PAUSE_LSW_FWD";
   IF #_w1 THEN "OP".HOOTER := TRUE; END_IF;
END_REGION

REGION Network 13: RET_LSW_UNHEATHY_POPOUP
   RUNG wire#powerrail
      Contact( "CYCLE_PAUSE_LSW_RET" )
      wire#w1
      Coil( "ALARM_12" )
   END_RUNG
   RUNG wire#w1
      P_Trig( "P_TRIG_11" )
      S_Coil( "OP".HOOTER )
   END_RUNG
   // the same network as SCL:
   "ALARM_12" := "CYCLE_PAUSE_LSW_RET";
   #_w1 := "CYCLE_PAUSE_LSW_RET" AND NOT "P_TRIG_11";   // rising edge
   "P_TRIG_11" := "CYCLE_PAUSE_LSW_RET";
   IF #_w1 THEN "OP".HOOTER := TRUE; END_IF;
END_REGION
END_FUNCTION

FUNCTION "LSW_INTERLOCK" : Void   // FC9, LAD
{ S7_Optimized_Access := 'TRUE' }
// stored: SetENOAutomatically false
   VAR_TEMP   // added for the SCL form of the ladder/FBD networks
      _w1 : Bool;
      _w2 : Bool;
   END_VAR
BEGIN

REGION Network 1: FORWARD LSW
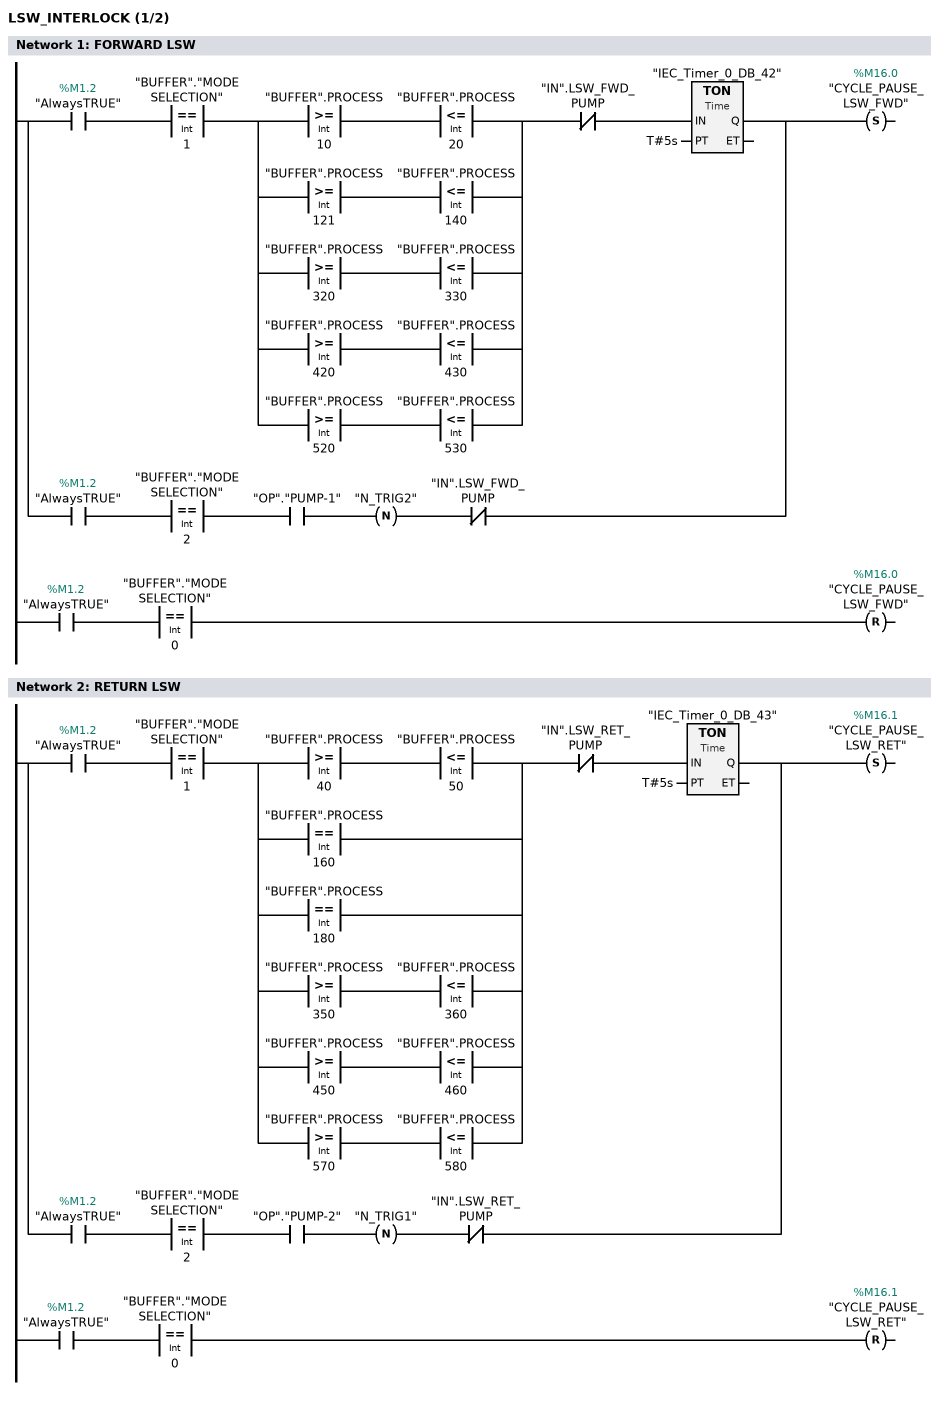
   RUNG wire#powerrail
      Contact( "AlwaysTRUE" )
      { S7_Templates := "SrcType := Int" } EQ_Contact(in1 := "BUFFER"."MODE SELECTION", in2 := 1)
      wire#w1
      { S7_Templates := "SrcType := Int" } GE_Contact(in1 := "BUFFER".PROCESS, in2 := 10)
      { S7_Templates := "SrcType := Int" } LE_Contact(in1 := "BUFFER".PROCESS, in2 := 20)
      wire#w2
      I_Contact( "IN".LSW_FWD_PUMP )
      { S7_Templates := "time_type := Time" } "IEC_Timer_0_DB_42".TON(pt := T#5s, et =>)
      wire#w3
      S_Coil( "CYCLE_PAUSE_LSW_FWD" )
   END_RUNG
   RUNG wire#w1
      { S7_Templates := "SrcType := Int" } GE_Contact(in1 := "BUFFER".PROCESS, in2 := 121)
      { S7_Templates := "SrcType := Int" } LE_Contact(in1 := "BUFFER".PROCESS, in2 := 140)
   END_RUNG wire#w2
   RUNG wire#w1
      { S7_Templates := "SrcType := Int" } GE_Contact(in1 := "BUFFER".PROCESS, in2 := 320)
      { S7_Templates := "SrcType := Int" } LE_Contact(in1 := "BUFFER".PROCESS, in2 := 330)
   END_RUNG wire#w2
   RUNG wire#w1
      { S7_Templates := "SrcType := Int" } GE_Contact(in1 := "BUFFER".PROCESS, in2 := 420)
      { S7_Templates := "SrcType := Int" } LE_Contact(in1 := "BUFFER".PROCESS, in2 := 430)
   END_RUNG wire#w2
   RUNG wire#w1
      { S7_Templates := "SrcType := Int" } GE_Contact(in1 := "BUFFER".PROCESS, in2 := 520)
      { S7_Templates := "SrcType := Int" } LE_Contact(in1 := "BUFFER".PROCESS, in2 := 530)
   END_RUNG wire#w2
   RUNG wire#powerrail
      Contact( "AlwaysTRUE" )
      { S7_Templates := "SrcType := Int" } EQ_Contact(in1 := "BUFFER"."MODE SELECTION", in2 := 2)
      Contact( "OP"."PUMP-1" )
      N_Trig( "N_TRIG2" )
      I_Contact( "IN".LSW_FWD_PUMP )
   END_RUNG wire#w3
   RUNG wire#powerrail
      Contact( "AlwaysTRUE" )
      { S7_Templates := "SrcType := Int" } EQ_Contact(in1 := "BUFFER"."MODE SELECTION", in2 := 0)
      R_Coil( "CYCLE_PAUSE_LSW_FWD" )
   END_RUNG
   // the same network as SCL:
   "IEC_Timer_0_DB_42".TON(IN := "AlwaysTRUE" AND ("BUFFER"."MODE SELECTION" = 1) AND ((("BUFFER".PROCESS >= 10) AND ("BUFFER".PROCESS <= 20)) OR (("BUFFER".PROCESS >= 121) AND ("BUFFER".PROCESS <= 140)) OR (("BUFFER".PROCESS >= 320) AND ("BUFFER".PROCESS <= 330)) OR (("BUFFER".PROCESS >= 420) AND ("BUFFER".PROCESS <= 430)) OR (("BUFFER".PROCESS >= 520) AND ("BUFFER".PROCESS <= 530))) AND NOT "IN".LSW_FWD_PUMP,
                           PT := T#5s);
   #_w1 := "AlwaysTRUE" AND ("BUFFER"."MODE SELECTION" = 2) AND "OP"."PUMP-1";
   #_w2 := NOT #_w1 AND "N_TRIG2";   // falling edge
   "N_TRIG2" := #_w1;
   IF "IEC_Timer_0_DB_42".Q OR (#_w2 AND NOT "IN".LSW_FWD_PUMP) THEN "CYCLE_PAUSE_LSW_FWD" := TRUE; END_IF;
   IF "AlwaysTRUE" AND ("BUFFER"."MODE SELECTION" = 0) THEN "CYCLE_PAUSE_LSW_FWD" := FALSE; END_IF;
END_REGION

REGION Network 2: RETURN LSW
   RUNG wire#powerrail
      Contact( "AlwaysTRUE" )
      { S7_Templates := "SrcType := Int" } EQ_Contact(in1 := "BUFFER"."MODE SELECTION", in2 := 1)
      wire#w1
      { S7_Templates := "SrcType := Int" } GE_Contact(in1 := "BUFFER".PROCESS, in2 := 40)
      { S7_Templates := "SrcType := Int" } LE_Contact(in1 := "BUFFER".PROCESS, in2 := 50)
      wire#w2
      I_Contact( "IN".LSW_RET_PUMP )
      { S7_Templates := "time_type := Time" } "IEC_Timer_0_DB_43".TON(pt := T#5s, et =>)
      wire#w3
      S_Coil( "CYCLE_PAUSE_LSW_RET" )
   END_RUNG
   RUNG wire#w1
      { S7_Templates := "SrcType := Int" } EQ_Contact(in1 := "BUFFER".PROCESS, in2 := 160)
   END_RUNG wire#w2
   RUNG wire#w1
      { S7_Templates := "SrcType := Int" } EQ_Contact(in1 := "BUFFER".PROCESS, in2 := 180)
   END_RUNG wire#w2
   RUNG wire#w1
      { S7_Templates := "SrcType := Int" } GE_Contact(in1 := "BUFFER".PROCESS, in2 := 350)
      { S7_Templates := "SrcType := Int" } LE_Contact(in1 := "BUFFER".PROCESS, in2 := 360)
   END_RUNG wire#w2
   RUNG wire#w1
      { S7_Templates := "SrcType := Int" } GE_Contact(in1 := "BUFFER".PROCESS, in2 := 450)
      { S7_Templates := "SrcType := Int" } LE_Contact(in1 := "BUFFER".PROCESS, in2 := 460)
   END_RUNG wire#w2
   RUNG wire#w1
      { S7_Templates := "SrcType := Int" } GE_Contact(in1 := "BUFFER".PROCESS, in2 := 570)
      { S7_Templates := "SrcType := Int" } LE_Contact(in1 := "BUFFER".PROCESS, in2 := 580)
   END_RUNG wire#w2
   RUNG wire#powerrail
      Contact( "AlwaysTRUE" )
      { S7_Templates := "SrcType := Int" } EQ_Contact(in1 := "BUFFER"."MODE SELECTION", in2 := 2)
      Contact( "OP"."PUMP-2" )
      N_Trig( "N_TRIG1" )
      I_Contact( "IN".LSW_RET_PUMP )
   END_RUNG wire#w3
   RUNG wire#powerrail
      Contact( "AlwaysTRUE" )
      { S7_Templates := "SrcType := Int" } EQ_Contact(in1 := "BUFFER"."MODE SELECTION", in2 := 0)
      R_Coil( "CYCLE_PAUSE_LSW_RET" )
   END_RUNG
   // the same network as SCL:
   "IEC_Timer_0_DB_43".TON(IN := "AlwaysTRUE" AND ("BUFFER"."MODE SELECTION" = 1) AND ((("BUFFER".PROCESS >= 40) AND ("BUFFER".PROCESS <= 50)) OR ("BUFFER".PROCESS = 160) OR ("BUFFER".PROCESS = 180) OR (("BUFFER".PROCESS >= 350) AND ("BUFFER".PROCESS <= 360)) OR (("BUFFER".PROCESS >= 450) AND ("BUFFER".PROCESS <= 460)) OR (("BUFFER".PROCESS >= 570) AND ("BUFFER".PROCESS <= 580))) AND NOT "IN".LSW_RET_PUMP,
                           PT := T#5s);
   #_w1 := "AlwaysTRUE" AND ("BUFFER"."MODE SELECTION" = 2) AND "OP"."PUMP-2";
   #_w2 := NOT #_w1 AND "N_TRIG1";   // falling edge
   "N_TRIG1" := #_w1;
   IF "IEC_Timer_0_DB_43".Q OR (#_w2 AND NOT "IN".LSW_RET_PUMP) THEN "CYCLE_PAUSE_LSW_RET" := TRUE; END_IF;
   IF "AlwaysTRUE" AND ("BUFFER"."MODE SELECTION" = 0) THEN "CYCLE_PAUSE_LSW_RET" := FALSE; END_IF;
END_REGION

REGION Network 3: cycle pause
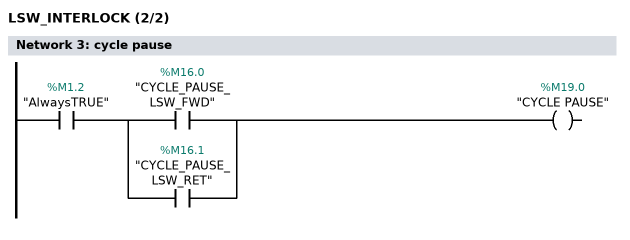
   RUNG wire#powerrail
      Contact( "AlwaysTRUE" )
      wire#w1
      Contact( "CYCLE_PAUSE_LSW_FWD" )
      wire#w2
      Coil( "CYCLE PAUSE" )
   END_RUNG
   RUNG wire#w1
      Contact( "CYCLE_PAUSE_LSW_RET" )
   END_RUNG wire#w2
   // the same network as SCL:
   "CYCLE PAUSE" := "AlwaysTRUE" AND ("CYCLE_PAUSE_LSW_FWD" OR "CYCLE_PAUSE_LSW_RET");
END_REGION
END_FUNCTION

DATA_BLOCK "CONDANSATE VALVE TIMER"   // DB33
// stored: InstanceOfName TIMING_BLOCK, InstanceOfType FB
"TIMING_BLOCK"
BEGIN
END_DATA_BLOCK

DATA_BLOCK "FINAL_RINSE_CONDUCTIVITY CHECK"   // DB4
// stored: InstanceOfName TIMING_BLOCK, InstanceOfType FB
"TIMING_BLOCK"
BEGIN
END_DATA_BLOCK

DATA_BLOCK "PW TANK_CLEANING"   // DB187
// stored: InstanceOfName TIMING_BLOCK, InstanceOfType FB
"TIMING_BLOCK"
BEGIN
END_DATA_BLOCK

DATA_BLOCK "PW TANK_DRAIN"   // DB188
// stored: InstanceOfName TIMING_BLOCK, InstanceOfType FB
"TIMING_BLOCK"
BEGIN
END_DATA_BLOCK

DATA_BLOCK "PW TANK_PUMP_CHASING"   // DB189
// stored: InstanceOfName TIMING_BLOCK, InstanceOfType FB
"TIMING_BLOCK"
BEGIN
END_DATA_BLOCK

DATA_BLOCK "PW TANK_PUMP_CHASING_1"   // DB207
// stored: InstanceOfName TIMING_BLOCK, InstanceOfType FB
"TIMING_BLOCK"
BEGIN
END_DATA_BLOCK

DATA_BLOCK "SCALE_DB_CT"   // DB25
// stored: InstanceOfName SCALE, InstanceOfType FB
"SCALE"
BEGIN
END_DATA_BLOCK

DATA_BLOCK "SCALE_DB_PH"   // DB8
// stored: InstanceOfName SCALE, InstanceOfType FB
"SCALE"
BEGIN
END_DATA_BLOCK

DATA_BLOCK "SCALE_DB_TT"   // DB6
// stored: InstanceOfName SCALE, InstanceOfType FB
"SCALE"
BEGIN
END_DATA_BLOCK

DATA_BLOCK "SW TANK_CLEANING"   // DB32
// stored: InstanceOfName TIMING_BLOCK, InstanceOfType FB
"TIMING_BLOCK"
BEGIN
END_DATA_BLOCK

DATA_BLOCK "SW TANK_DRAIN"   // DB182
// stored: InstanceOfName TIMING_BLOCK, InstanceOfType FB
"TIMING_BLOCK"
BEGIN
END_DATA_BLOCK

DATA_BLOCK "SW TANK_PUMP_CHASING"   // DB186
// stored: InstanceOfName TIMING_BLOCK, InstanceOfType FB
"TIMING_BLOCK"
BEGIN
END_DATA_BLOCK

DATA_BLOCK "SW TANK_PUMP_CHASING_1"   // DB209
// stored: InstanceOfName TIMING_BLOCK, InstanceOfType FB
"TIMING_BLOCK"
BEGIN
END_DATA_BLOCK

DATA_BLOCK "TIMING_BLOCK_DB"   // DB198
// stored: InstanceOfName TIMING_BLOCK, InstanceOfType FB
"TIMING_BLOCK"
BEGIN
END_DATA_BLOCK

DATA_BLOCK "start dosing and recirculation_DB_1"   // DB190
// stored: InstanceOfName TIMING_BLOCK, InstanceOfType FB
"TIMING_BLOCK"
BEGIN
END_DATA_BLOCK

DATA_BLOCK "ACID_DOSING"   // DB59
// stored: InstanceOfName TIMING_BLOCK, InstanceOfType FB
"TIMING_BLOCK"
BEGIN
END_DATA_BLOCK

DATA_BLOCK "DOSING"   // DB57
// stored: InstanceOfName TIMING_BLOCK, InstanceOfType FB
"TIMING_BLOCK"
BEGIN
END_DATA_BLOCK

DATA_BLOCK "FINAL_RINSE_CLEANING"   // DB71
// stored: InstanceOfName TIMING_BLOCK, InstanceOfType FB
"TIMING_BLOCK"
BEGIN
END_DATA_BLOCK

DATA_BLOCK "FINAL_RINSE_DRAIN"   // DB90
// stored: InstanceOfName TIMING_BLOCK, InstanceOfType FB
"TIMING_BLOCK"
BEGIN
END_DATA_BLOCK

DATA_BLOCK "FINAL_RINSE_PUMP_CHASING"   // DB93
// stored: InstanceOfName TIMING_BLOCK, InstanceOfType FB
"TIMING_BLOCK"
BEGIN
END_DATA_BLOCK

DATA_BLOCK "FINAL_RINSE_RECIRCULATION"   // DB88
// stored: InstanceOfName TIMING_BLOCK, InstanceOfType FB
"TIMING_BLOCK"
BEGIN
END_DATA_BLOCK

DATA_BLOCK "RINSE-1_CLEANING"   // DB7
// stored: InstanceOfName TIMING_BLOCK, InstanceOfType FB
"TIMING_BLOCK"
BEGIN
END_DATA_BLOCK

DATA_BLOCK "RINSE-1_DRAIN"   // DB42
// stored: InstanceOfName TIMING_BLOCK, InstanceOfType FB
"TIMING_BLOCK"
BEGIN
END_DATA_BLOCK

DATA_BLOCK "RINSE-1_PUMP_CHASING"   // DB44
// stored: InstanceOfName TIMING_BLOCK, InstanceOfType FB
"TIMING_BLOCK"
BEGIN
END_DATA_BLOCK

DATA_BLOCK "RINSE-1_RECIRCULATION"   // DB40
// stored: InstanceOfName TIMING_BLOCK, InstanceOfType FB
"TIMING_BLOCK"
BEGIN
END_DATA_BLOCK

DATA_BLOCK "RINSE-2_CLEANING"   // DB48
// stored: InstanceOfName TIMING_BLOCK, InstanceOfType FB
"TIMING_BLOCK"
BEGIN
END_DATA_BLOCK

DATA_BLOCK "RINSE-2_DRAIN"   // DB52
// stored: InstanceOfName TIMING_BLOCK, InstanceOfType FB
"TIMING_BLOCK"
BEGIN
END_DATA_BLOCK

DATA_BLOCK "RINSE-2_PUMP_CHASING"   // DB54
// stored: InstanceOfName TIMING_BLOCK, InstanceOfType FB
"TIMING_BLOCK"
BEGIN
END_DATA_BLOCK

DATA_BLOCK "RINSE-2_RECIRCULATION"   // DB50
// stored: InstanceOfName TIMING_BLOCK, InstanceOfType FB
"TIMING_BLOCK"
BEGIN
END_DATA_BLOCK

DATA_BLOCK "RINSE-3_CLEANING"   // DB78
// stored: InstanceOfName TIMING_BLOCK, InstanceOfType FB
"TIMING_BLOCK"
BEGIN
END_DATA_BLOCK

DATA_BLOCK "RINSE-3_DRAIN"   // DB81
// stored: InstanceOfName TIMING_BLOCK, InstanceOfType FB
"TIMING_BLOCK"
BEGIN
END_DATA_BLOCK

DATA_BLOCK "RINSE-3_PUMP_CHASING"   // DB83
// stored: InstanceOfName TIMING_BLOCK, InstanceOfType FB
"TIMING_BLOCK"
BEGIN
END_DATA_BLOCK

DATA_BLOCK "RINSE-3_RECIRCULATION"   // DB79
// stored: InstanceOfName TIMING_BLOCK, InstanceOfType FB
"TIMING_BLOCK"
BEGIN
END_DATA_BLOCK

DATA_BLOCK "IEC_Timer_0_DB_1"   // DB39
{ S7_Optimized_Access := 'TRUE' }
// stored: InstanceOfName IEC_TIMER, OfSystemLibElement IEC_TIMER, OfSystemLibVersion 1.0
"IEC_TIMER"
   // VAR
   //    PT : Time;
   //    ET { ExternalWritable := 'False'} : Time;
   //    IN : Bool;
   //    Q { ExternalWritable := 'False'} : Bool;
   // END_VAR
BEGIN
END_DATA_BLOCK

DATA_BLOCK "IEC_Timer_0_DB_10"   // DB55
{ S7_Optimized_Access := 'TRUE' }
// stored: InstanceOfName IEC_TIMER, OfSystemLibElement IEC_TIMER, OfSystemLibVersion 1.0
"IEC_TIMER"
   // VAR
   //    PT : Time;
   //    ET { ExternalWritable := 'False'} : Time;
   //    IN : Bool;
   //    Q { ExternalWritable := 'False'} : Bool;
   // END_VAR
BEGIN
END_DATA_BLOCK

DATA_BLOCK "IEC_Timer_0_DB_11"   // DB56
{ S7_Optimized_Access := 'TRUE' }
// stored: InstanceOfName IEC_TIMER, OfSystemLibElement IEC_TIMER, OfSystemLibVersion 1.0
"IEC_TIMER"
   // VAR
   //    PT : Time;
   //    ET { ExternalWritable := 'False'} : Time;
   //    IN : Bool;
   //    Q { ExternalWritable := 'False'} : Bool;
   // END_VAR
BEGIN
END_DATA_BLOCK

DATA_BLOCK "IEC_Timer_0_DB_12"   // DB15
{ S7_Optimized_Access := 'TRUE' }
// stored: InstanceOfName IEC_TIMER, OfSystemLibElement IEC_TIMER, OfSystemLibVersion 1.0
"IEC_TIMER"
   // VAR
   //    PT : Time;
   //    ET { ExternalWritable := 'False'} : Time;
   //    IN : Bool;
   //    Q { ExternalWritable := 'False'} : Bool;
   // END_VAR
BEGIN
END_DATA_BLOCK

DATA_BLOCK "IEC_Timer_0_DB_120"   // DB191
{ S7_Optimized_Access := 'TRUE' }
// stored: InstanceOfName IEC_TIMER, OfSystemLibElement IEC_TIMER, OfSystemLibVersion 1.0
"IEC_TIMER"
   // VAR
   //    PT : Time;
   //    ET { ExternalWritable := 'False'} : Time;
   //    IN : Bool;
   //    Q { ExternalWritable := 'False'} : Bool;
   // END_VAR
BEGIN
END_DATA_BLOCK

DATA_BLOCK "IEC_Timer_0_DB_124"   // DB192
{ S7_Optimized_Access := 'TRUE' }
// stored: InstanceOfName IEC_TIMER, OfSystemLibElement IEC_TIMER, OfSystemLibVersion 1.0
"IEC_TIMER"
   // VAR
   //    PT : Time;
   //    ET { ExternalWritable := 'False'} : Time;
   //    IN : Bool;
   //    Q { ExternalWritable := 'False'} : Bool;
   // END_VAR
BEGIN
END_DATA_BLOCK

DATA_BLOCK "IEC_Timer_0_DB_125"   // DB193
{ S7_Optimized_Access := 'TRUE' }
// stored: InstanceOfName IEC_TIMER, OfSystemLibElement IEC_TIMER, OfSystemLibVersion 1.0
"IEC_TIMER"
   // VAR
   //    PT : Time;
   //    ET { ExternalWritable := 'False'} : Time;
   //    IN : Bool;
   //    Q { ExternalWritable := 'False'} : Bool;
   // END_VAR
BEGIN
END_DATA_BLOCK

DATA_BLOCK "IEC_Timer_0_DB_126"   // DB194
{ S7_Optimized_Access := 'TRUE' }
// stored: InstanceOfName IEC_TIMER, OfSystemLibElement IEC_TIMER, OfSystemLibVersion 1.0
"IEC_TIMER"
   // VAR
   //    PT : Time;
   //    ET { ExternalWritable := 'False'} : Time;
   //    IN : Bool;
   //    Q { ExternalWritable := 'False'} : Bool;
   // END_VAR
BEGIN
END_DATA_BLOCK

DATA_BLOCK "IEC_Timer_0_DB_127"   // DB195
{ S7_Optimized_Access := 'TRUE' }
// stored: InstanceOfName IEC_TIMER, OfSystemLibElement IEC_TIMER, OfSystemLibVersion 1.0
"IEC_TIMER"
   // VAR
   //    PT : Time;
   //    ET { ExternalWritable := 'False'} : Time;
   //    IN : Bool;
   //    Q { ExternalWritable := 'False'} : Bool;
   // END_VAR
BEGIN
END_DATA_BLOCK

DATA_BLOCK "IEC_Timer_0_DB_128"   // DB196
{ S7_Optimized_Access := 'TRUE' }
// stored: InstanceOfName IEC_TIMER, OfSystemLibElement IEC_TIMER, OfSystemLibVersion 1.0
"IEC_TIMER"
   // VAR
   //    PT : Time;
   //    ET { ExternalWritable := 'False'} : Time;
   //    IN : Bool;
   //    Q { ExternalWritable := 'False'} : Bool;
   // END_VAR
BEGIN
END_DATA_BLOCK

DATA_BLOCK "IEC_Timer_0_DB_129"   // DB197
{ S7_Optimized_Access := 'TRUE' }
// stored: InstanceOfName IEC_TIMER, OfSystemLibElement IEC_TIMER, OfSystemLibVersion 1.0
"IEC_TIMER"
   // VAR
   //    PT : Time;
   //    ET { ExternalWritable := 'False'} : Time;
   //    IN : Bool;
   //    Q { ExternalWritable := 'False'} : Bool;
   // END_VAR
BEGIN
END_DATA_BLOCK

DATA_BLOCK "IEC_Timer_0_DB_13"   // DB14
{ S7_Optimized_Access := 'TRUE' }
// stored: InstanceOfName IEC_TIMER, OfSystemLibElement IEC_TIMER, OfSystemLibVersion 1.0
"IEC_TIMER"
   // VAR
   //    PT : Time;
   //    ET { ExternalWritable := 'False'} : Time;
   //    IN : Bool;
   //    Q { ExternalWritable := 'False'} : Bool;
   // END_VAR
BEGIN
END_DATA_BLOCK

DATA_BLOCK "IEC_Timer_0_DB_130"   // DB199
{ S7_Optimized_Access := 'TRUE' }
// stored: InstanceOfName IEC_TIMER, OfSystemLibElement IEC_TIMER, OfSystemLibVersion 1.0
"IEC_TIMER"
   // VAR
   //    PT : Time;
   //    ET { ExternalWritable := 'False'} : Time;
   //    IN : Bool;
   //    Q { ExternalWritable := 'False'} : Bool;
   // END_VAR
BEGIN
END_DATA_BLOCK

DATA_BLOCK "IEC_Timer_0_DB_131"   // DB200
{ S7_Optimized_Access := 'TRUE' }
// stored: InstanceOfName IEC_TIMER, OfSystemLibElement IEC_TIMER, OfSystemLibVersion 1.0
"IEC_TIMER"
   // VAR
   //    PT : Time;
   //    ET { ExternalWritable := 'False'} : Time;
   //    IN : Bool;
   //    Q { ExternalWritable := 'False'} : Bool;
   // END_VAR
BEGIN
END_DATA_BLOCK

DATA_BLOCK "IEC_Timer_0_DB_132"   // DB201
{ S7_Optimized_Access := 'TRUE' }
// stored: InstanceOfName IEC_TIMER, OfSystemLibElement IEC_TIMER, OfSystemLibVersion 1.0
"IEC_TIMER"
   // VAR
   //    PT : Time;
   //    ET { ExternalWritable := 'False'} : Time;
   //    IN : Bool;
   //    Q { ExternalWritable := 'False'} : Bool;
   // END_VAR
BEGIN
END_DATA_BLOCK

DATA_BLOCK "IEC_Timer_0_DB_133"   // DB202
{ S7_Optimized_Access := 'TRUE' }
// stored: InstanceOfName IEC_TIMER, OfSystemLibElement IEC_TIMER, OfSystemLibVersion 1.0
"IEC_TIMER"
   // VAR
   //    PT : Time;
   //    ET { ExternalWritable := 'False'} : Time;
   //    IN : Bool;
   //    Q { ExternalWritable := 'False'} : Bool;
   // END_VAR
BEGIN
END_DATA_BLOCK

DATA_BLOCK "IEC_Timer_0_DB_134"   // DB203
{ S7_Optimized_Access := 'TRUE' }
// stored: InstanceOfName IEC_TIMER, OfSystemLibElement IEC_TIMER, OfSystemLibVersion 1.0
"IEC_TIMER"
   // VAR
   //    PT : Time;
   //    ET { ExternalWritable := 'False'} : Time;
   //    IN : Bool;
   //    Q { ExternalWritable := 'False'} : Bool;
   // END_VAR
BEGIN
END_DATA_BLOCK

DATA_BLOCK "IEC_Timer_0_DB_135"   // DB204
{ S7_Optimized_Access := 'TRUE' }
// stored: InstanceOfName IEC_TIMER, OfSystemLibElement IEC_TIMER, OfSystemLibVersion 1.0
"IEC_TIMER"
   // VAR
   //    PT : Time;
   //    ET { ExternalWritable := 'False'} : Time;
   //    IN : Bool;
   //    Q { ExternalWritable := 'False'} : Bool;
   // END_VAR
BEGIN
END_DATA_BLOCK

DATA_BLOCK "IEC_Timer_0_DB_136"   // DB205
{ S7_Optimized_Access := 'TRUE' }
// stored: InstanceOfName IEC_TIMER, OfSystemLibElement IEC_TIMER, OfSystemLibVersion 1.0
"IEC_TIMER"
   // VAR
   //    PT : Time;
   //    ET { ExternalWritable := 'False'} : Time;
   //    IN : Bool;
   //    Q { ExternalWritable := 'False'} : Bool;
   // END_VAR
BEGIN
END_DATA_BLOCK

DATA_BLOCK "IEC_Timer_0_DB_137"   // DB208
{ S7_Optimized_Access := 'TRUE' }
// stored: InstanceOfName IEC_TIMER, OfSystemLibElement IEC_TIMER, OfSystemLibVersion 1.0
"IEC_TIMER"
   // VAR
   //    PT : Time;
   //    ET { ExternalWritable := 'False'} : Time;
   //    IN : Bool;
   //    Q { ExternalWritable := 'False'} : Bool;
   // END_VAR
BEGIN
END_DATA_BLOCK

DATA_BLOCK "IEC_Timer_0_DB_139"   // DB212
{ S7_Optimized_Access := 'TRUE' }
// stored: InstanceOfName IEC_TIMER, OfSystemLibElement IEC_TIMER, OfSystemLibVersion 1.0
"IEC_TIMER"
   // VAR
   //    PT : Time;
   //    ET { ExternalWritable := 'False'} : Time;
   //    IN : Bool;
   //    Q { ExternalWritable := 'False'} : Bool;
   // END_VAR
BEGIN
END_DATA_BLOCK

DATA_BLOCK "IEC_Timer_0_DB_14"   // DB61
{ S7_Optimized_Access := 'TRUE' }
// stored: InstanceOfName IEC_TIMER, OfSystemLibElement IEC_TIMER, OfSystemLibVersion 1.0
"IEC_TIMER"
   // VAR
   //    PT : Time;
   //    ET { ExternalWritable := 'False'} : Time;
   //    IN : Bool;
   //    Q { ExternalWritable := 'False'} : Bool;
   // END_VAR
BEGIN
END_DATA_BLOCK

DATA_BLOCK "IEC_Timer_0_DB_140"   // DB213
{ S7_Optimized_Access := 'TRUE' }
// stored: InstanceOfName IEC_TIMER, OfSystemLibElement IEC_TIMER, OfSystemLibVersion 1.0
"IEC_TIMER"
   // VAR
   //    PT : Time;
   //    ET { ExternalWritable := 'False'} : Time;
   //    IN : Bool;
   //    Q { ExternalWritable := 'False'} : Bool;
   // END_VAR
BEGIN
END_DATA_BLOCK

DATA_BLOCK "IEC_Timer_0_DB_141"   // DB214
{ S7_Optimized_Access := 'TRUE' }
// stored: InstanceOfName IEC_TIMER, OfSystemLibElement IEC_TIMER, OfSystemLibVersion 1.0
"IEC_TIMER"
   // VAR
   //    PT : Time;
   //    ET { ExternalWritable := 'False'} : Time;
   //    IN : Bool;
   //    Q { ExternalWritable := 'False'} : Bool;
   // END_VAR
BEGIN
END_DATA_BLOCK

DATA_BLOCK "IEC_Timer_0_DB_142"   // DB215
{ S7_Optimized_Access := 'TRUE' }
// stored: InstanceOfName IEC_TIMER, OfSystemLibElement IEC_TIMER, OfSystemLibVersion 1.0
"IEC_TIMER"
   // VAR
   //    PT : Time;
   //    ET { ExternalWritable := 'False'} : Time;
   //    IN : Bool;
   //    Q { ExternalWritable := 'False'} : Bool;
   // END_VAR
BEGIN
END_DATA_BLOCK

DATA_BLOCK "IEC_Timer_0_DB_143"   // DB216
{ S7_Optimized_Access := 'TRUE' }
// stored: InstanceOfName IEC_TIMER, OfSystemLibElement IEC_TIMER, OfSystemLibVersion 1.0
"IEC_TIMER"
   // VAR
   //    PT : Time;
   //    ET { ExternalWritable := 'False'} : Time;
   //    IN : Bool;
   //    Q { ExternalWritable := 'False'} : Bool;
   // END_VAR
BEGIN
END_DATA_BLOCK

DATA_BLOCK "IEC_Timer_0_DB_15"   // DB63
{ S7_Optimized_Access := 'TRUE' }
// stored: InstanceOfName IEC_TIMER, OfSystemLibElement IEC_TIMER, OfSystemLibVersion 1.0
"IEC_TIMER"
   // VAR
   //    PT : Time;
   //    ET { ExternalWritable := 'False'} : Time;
   //    IN : Bool;
   //    Q { ExternalWritable := 'False'} : Bool;
   // END_VAR
BEGIN
END_DATA_BLOCK

DATA_BLOCK "IEC_Timer_0_DB_16"   // DB65
{ S7_Optimized_Access := 'TRUE' }
// stored: InstanceOfName IEC_TIMER, OfSystemLibElement IEC_TIMER, OfSystemLibVersion 1.0
"IEC_TIMER"
   // VAR
   //    PT : Time;
   //    ET { ExternalWritable := 'False'} : Time;
   //    IN : Bool;
   //    Q { ExternalWritable := 'False'} : Bool;
   // END_VAR
BEGIN
END_DATA_BLOCK

DATA_BLOCK "IEC_Timer_0_DB_17"   // DB67
{ S7_Optimized_Access := 'TRUE' }
// stored: InstanceOfName IEC_TIMER, OfSystemLibElement IEC_TIMER, OfSystemLibVersion 1.0
"IEC_TIMER"
   // VAR
   //    PT : Time;
   //    ET { ExternalWritable := 'False'} : Time;
   //    IN : Bool;
   //    Q { ExternalWritable := 'False'} : Bool;
   // END_VAR
BEGIN
END_DATA_BLOCK

DATA_BLOCK "IEC_Timer_0_DB_18"   // DB69
{ S7_Optimized_Access := 'TRUE' }
// stored: InstanceOfName IEC_TIMER, OfSystemLibElement IEC_TIMER, OfSystemLibVersion 1.0
"IEC_TIMER"
   // VAR
   //    PT : Time;
   //    ET { ExternalWritable := 'False'} : Time;
   //    IN : Bool;
   //    Q { ExternalWritable := 'False'} : Bool;
   // END_VAR
BEGIN
END_DATA_BLOCK

DATA_BLOCK "IEC_Timer_0_DB_19"   // DB12
{ S7_Optimized_Access := 'TRUE' }
// stored: InstanceOfName IEC_TIMER, OfSystemLibElement IEC_TIMER, OfSystemLibVersion 1.0
"IEC_TIMER"
   // VAR
   //    PT : Time;
   //    ET { ExternalWritable := 'False'} : Time;
   //    IN : Bool;
   //    Q { ExternalWritable := 'False'} : Bool;
   // END_VAR
BEGIN
END_DATA_BLOCK

DATA_BLOCK "IEC_Timer_0_DB_2"   // DB41
{ S7_Optimized_Access := 'TRUE' }
// stored: InstanceOfName IEC_TIMER, OfSystemLibElement IEC_TIMER, OfSystemLibVersion 1.0
"IEC_TIMER"
   // VAR
   //    PT : Time;
   //    ET { ExternalWritable := 'False'} : Time;
   //    IN : Bool;
   //    Q { ExternalWritable := 'False'} : Bool;
   // END_VAR
BEGIN
END_DATA_BLOCK

DATA_BLOCK "IEC_Timer_0_DB_20"   // DB72
{ S7_Optimized_Access := 'TRUE' }
// stored: InstanceOfName IEC_TIMER, OfSystemLibElement IEC_TIMER, OfSystemLibVersion 1.0
"IEC_TIMER"
   // VAR
   //    PT : Time;
   //    ET { ExternalWritable := 'False'} : Time;
   //    IN : Bool;
   //    Q { ExternalWritable := 'False'} : Bool;
   // END_VAR
BEGIN
END_DATA_BLOCK

DATA_BLOCK "IEC_Timer_0_DB_21"   // DB2
{ S7_Optimized_Access := 'TRUE' }
// stored: InstanceOfName IEC_TIMER, OfSystemLibElement IEC_TIMER, OfSystemLibVersion 1.0
"IEC_TIMER"
   // VAR
   //    PT : Time;
   //    ET { ExternalWritable := 'False'} : Time;
   //    IN : Bool;
   //    Q { ExternalWritable := 'False'} : Bool;
   // END_VAR
BEGIN
END_DATA_BLOCK

DATA_BLOCK "IEC_Timer_0_DB_22"   // DB3
{ S7_Optimized_Access := 'TRUE' }
// stored: InstanceOfName IEC_TIMER, OfSystemLibElement IEC_TIMER, OfSystemLibVersion 1.0
"IEC_TIMER"
   // VAR
   //    PT : Time;
   //    ET { ExternalWritable := 'False'} : Time;
   //    IN : Bool;
   //    Q { ExternalWritable := 'False'} : Bool;
   // END_VAR
BEGIN
END_DATA_BLOCK

DATA_BLOCK "IEC_Timer_0_DB_23"   // DB16
{ S7_Optimized_Access := 'TRUE' }
// stored: InstanceOfName IEC_TIMER, OfSystemLibElement IEC_TIMER, OfSystemLibVersion 1.0
"IEC_TIMER"
   // VAR
   //    PT : Time;
   //    ET { ExternalWritable := 'False'} : Time;
   //    IN : Bool;
   //    Q { ExternalWritable := 'False'} : Bool;
   // END_VAR
BEGIN
END_DATA_BLOCK

DATA_BLOCK "IEC_Timer_0_DB_24"   // DB17
{ S7_Optimized_Access := 'TRUE' }
// stored: InstanceOfName IEC_TIMER, OfSystemLibElement IEC_TIMER, OfSystemLibVersion 1.0
"IEC_TIMER"
   // VAR
   //    PT : Time;
   //    ET { ExternalWritable := 'False'} : Time;
   //    IN : Bool;
   //    Q { ExternalWritable := 'False'} : Bool;
   // END_VAR
BEGIN
END_DATA_BLOCK

DATA_BLOCK "IEC_Timer_0_DB_25"   // DB74
{ S7_Optimized_Access := 'TRUE' }
// stored: InstanceOfName IEC_TIMER, OfSystemLibElement IEC_TIMER, OfSystemLibVersion 1.0
"IEC_TIMER"
   // VAR
   //    PT : Time;
   //    ET { ExternalWritable := 'False'} : Time;
   //    IN : Bool;
   //    Q { ExternalWritable := 'False'} : Bool;
   // END_VAR
BEGIN
END_DATA_BLOCK

DATA_BLOCK "IEC_Timer_0_DB_26"   // DB75
{ S7_Optimized_Access := 'TRUE' }
// stored: InstanceOfName IEC_TIMER, OfSystemLibElement IEC_TIMER, OfSystemLibVersion 1.0
"IEC_TIMER"
   // VAR
   //    PT : Time;
   //    ET { ExternalWritable := 'False'} : Time;
   //    IN : Bool;
   //    Q { ExternalWritable := 'False'} : Bool;
   // END_VAR
BEGIN
END_DATA_BLOCK

DATA_BLOCK "IEC_Timer_0_DB_27"   // DB76
{ S7_Optimized_Access := 'TRUE' }
// stored: InstanceOfName IEC_TIMER, OfSystemLibElement IEC_TIMER, OfSystemLibVersion 1.0
"IEC_TIMER"
   // VAR
   //    PT : Time;
   //    ET { ExternalWritable := 'False'} : Time;
   //    IN : Bool;
   //    Q { ExternalWritable := 'False'} : Bool;
   // END_VAR
BEGIN
END_DATA_BLOCK

DATA_BLOCK "IEC_Timer_0_DB_28"   // DB77
{ S7_Optimized_Access := 'TRUE' }
// stored: InstanceOfName IEC_TIMER, OfSystemLibElement IEC_TIMER, OfSystemLibVersion 1.0
"IEC_TIMER"
   // VAR
   //    PT : Time;
   //    ET { ExternalWritable := 'False'} : Time;
   //    IN : Bool;
   //    Q { ExternalWritable := 'False'} : Bool;
   // END_VAR
BEGIN
END_DATA_BLOCK

DATA_BLOCK "IEC_Timer_0_DB_29"   // DB80
{ S7_Optimized_Access := 'TRUE' }
// stored: InstanceOfName IEC_TIMER, OfSystemLibElement IEC_TIMER, OfSystemLibVersion 1.0
"IEC_TIMER"
   // VAR
   //    PT : Time;
   //    ET { ExternalWritable := 'False'} : Time;
   //    IN : Bool;
   //    Q { ExternalWritable := 'False'} : Bool;
   // END_VAR
BEGIN
END_DATA_BLOCK

DATA_BLOCK "IEC_Timer_0_DB_3"   // DB43
{ S7_Optimized_Access := 'TRUE' }
// stored: InstanceOfName IEC_TIMER, OfSystemLibElement IEC_TIMER, OfSystemLibVersion 1.0
"IEC_TIMER"
   // VAR
   //    PT : Time;
   //    ET { ExternalWritable := 'False'} : Time;
   //    IN : Bool;
   //    Q { ExternalWritable := 'False'} : Bool;
   // END_VAR
BEGIN
END_DATA_BLOCK

DATA_BLOCK "IEC_Timer_0_DB_30"   // DB82
{ S7_Optimized_Access := 'TRUE' }
// stored: InstanceOfName IEC_TIMER, OfSystemLibElement IEC_TIMER, OfSystemLibVersion 1.0
"IEC_TIMER"
   // VAR
   //    PT : Time;
   //    ET { ExternalWritable := 'False'} : Time;
   //    IN : Bool;
   //    Q { ExternalWritable := 'False'} : Bool;
   // END_VAR
BEGIN
END_DATA_BLOCK

DATA_BLOCK "IEC_Timer_0_DB_31"   // DB84
{ S7_Optimized_Access := 'TRUE' }
// stored: InstanceOfName IEC_TIMER, OfSystemLibElement IEC_TIMER, OfSystemLibVersion 1.0
"IEC_TIMER"
   // VAR
   //    PT : Time;
   //    ET { ExternalWritable := 'False'} : Time;
   //    IN : Bool;
   //    Q { ExternalWritable := 'False'} : Bool;
   // END_VAR
BEGIN
END_DATA_BLOCK

DATA_BLOCK "IEC_Timer_0_DB_32"   // DB18
{ S7_Optimized_Access := 'TRUE' }
// stored: InstanceOfName IEC_TIMER, OfSystemLibElement IEC_TIMER, OfSystemLibVersion 1.0
"IEC_TIMER"
   // VAR
   //    PT : Time;
   //    ET { ExternalWritable := 'False'} : Time;
   //    IN : Bool;
   //    Q { ExternalWritable := 'False'} : Bool;
   // END_VAR
BEGIN
END_DATA_BLOCK

DATA_BLOCK "IEC_Timer_0_DB_33"   // DB89
{ S7_Optimized_Access := 'TRUE' }
// stored: InstanceOfName IEC_TIMER, OfSystemLibElement IEC_TIMER, OfSystemLibVersion 1.0
"IEC_TIMER"
   // VAR
   //    PT : Time;
   //    ET { ExternalWritable := 'False'} : Time;
   //    IN : Bool;
   //    Q { ExternalWritable := 'False'} : Bool;
   // END_VAR
BEGIN
END_DATA_BLOCK

DATA_BLOCK "IEC_Timer_0_DB_34"   // DB91
{ S7_Optimized_Access := 'TRUE' }
// stored: InstanceOfName IEC_TIMER, OfSystemLibElement IEC_TIMER, OfSystemLibVersion 1.0
"IEC_TIMER"
   // VAR
   //    PT : Time;
   //    ET { ExternalWritable := 'False'} : Time;
   //    IN : Bool;
   //    Q { ExternalWritable := 'False'} : Bool;
   // END_VAR
BEGIN
END_DATA_BLOCK

DATA_BLOCK "IEC_Timer_0_DB_35"   // DB92
{ S7_Optimized_Access := 'TRUE' }
// stored: InstanceOfName IEC_TIMER, OfSystemLibElement IEC_TIMER, OfSystemLibVersion 1.0
"IEC_TIMER"
   // VAR
   //    PT : Time;
   //    ET { ExternalWritable := 'False'} : Time;
   //    IN : Bool;
   //    Q { ExternalWritable := 'False'} : Bool;
   // END_VAR
BEGIN
END_DATA_BLOCK

DATA_BLOCK "IEC_Timer_0_DB_36"   // DB94
{ S7_Optimized_Access := 'TRUE' }
// stored: InstanceOfName IEC_TIMER, OfSystemLibElement IEC_TIMER, OfSystemLibVersion 1.0
"IEC_TIMER"
   // VAR
   //    PT : Time;
   //    ET { ExternalWritable := 'False'} : Time;
   //    IN : Bool;
   //    Q { ExternalWritable := 'False'} : Bool;
   // END_VAR
BEGIN
END_DATA_BLOCK

DATA_BLOCK "IEC_Timer_0_DB_37"   // DB95
{ S7_Optimized_Access := 'TRUE' }
// stored: InstanceOfName IEC_TIMER, OfSystemLibElement IEC_TIMER, OfSystemLibVersion 1.0
"IEC_TIMER"
   // VAR
   //    PT : Time;
   //    ET { ExternalWritable := 'False'} : Time;
   //    IN : Bool;
   //    Q { ExternalWritable := 'False'} : Bool;
   // END_VAR
BEGIN
END_DATA_BLOCK

DATA_BLOCK "IEC_Timer_0_DB_38"   // DB96
{ S7_Optimized_Access := 'TRUE' }
// stored: InstanceOfName IEC_TIMER, OfSystemLibElement IEC_TIMER, OfSystemLibVersion 1.0
"IEC_TIMER"
   // VAR
   //    PT : Time;
   //    ET { ExternalWritable := 'False'} : Time;
   //    IN : Bool;
   //    Q { ExternalWritable := 'False'} : Bool;
   // END_VAR
BEGIN
END_DATA_BLOCK

DATA_BLOCK "IEC_Timer_0_DB_39"   // DB13
{ S7_Optimized_Access := 'TRUE' }
// stored: InstanceOfName IEC_TIMER, OfSystemLibElement IEC_TIMER, OfSystemLibVersion 1.0
"IEC_TIMER"
   // VAR
   //    PT : Time;
   //    ET { ExternalWritable := 'False'} : Time;
   //    IN : Bool;
   //    Q { ExternalWritable := 'False'} : Bool;
   // END_VAR
BEGIN
END_DATA_BLOCK

DATA_BLOCK "IEC_Timer_0_DB_4"   // DB45
{ S7_Optimized_Access := 'TRUE' }
// stored: InstanceOfName IEC_TIMER, OfSystemLibElement IEC_TIMER, OfSystemLibVersion 1.0
"IEC_TIMER"
   // VAR
   //    PT : Time;
   //    ET { ExternalWritable := 'False'} : Time;
   //    IN : Bool;
   //    Q { ExternalWritable := 'False'} : Bool;
   // END_VAR
BEGIN
END_DATA_BLOCK

DATA_BLOCK "IEC_Timer_0_DB_40"   // DB19
{ S7_Optimized_Access := 'TRUE' }
// stored: InstanceOfName IEC_TIMER, OfSystemLibElement IEC_TIMER, OfSystemLibVersion 1.0
"IEC_TIMER"
   // VAR
   //    PT : Time;
   //    ET { ExternalWritable := 'False'} : Time;
   //    IN : Bool;
   //    Q { ExternalWritable := 'False'} : Bool;
   // END_VAR
BEGIN
END_DATA_BLOCK

DATA_BLOCK "IEC_Timer_0_DB_41"   // DB20
{ S7_Optimized_Access := 'TRUE' }
// stored: InstanceOfName IEC_TIMER, OfSystemLibElement IEC_TIMER, OfSystemLibVersion 1.0
"IEC_TIMER"
   // VAR
   //    PT : Time;
   //    ET { ExternalWritable := 'False'} : Time;
   //    IN : Bool;
   //    Q { ExternalWritable := 'False'} : Bool;
   // END_VAR
BEGIN
END_DATA_BLOCK

DATA_BLOCK "IEC_Timer_0_DB_42"   // DB21
{ S7_Optimized_Access := 'TRUE' }
// stored: InstanceOfName IEC_TIMER, OfSystemLibElement IEC_TIMER, OfSystemLibVersion 1.0
"IEC_TIMER"
   // VAR
   //    PT : Time;
   //    ET { ExternalWritable := 'False'} : Time;
   //    IN : Bool;
   //    Q { ExternalWritable := 'False'} : Bool;
   // END_VAR
BEGIN
END_DATA_BLOCK

DATA_BLOCK "IEC_Timer_0_DB_43"   // DB22
{ S7_Optimized_Access := 'TRUE' }
// stored: InstanceOfName IEC_TIMER, OfSystemLibElement IEC_TIMER, OfSystemLibVersion 1.0
"IEC_TIMER"
   // VAR
   //    PT : Time;
   //    ET { ExternalWritable := 'False'} : Time;
   //    IN : Bool;
   //    Q { ExternalWritable := 'False'} : Bool;
   // END_VAR
BEGIN
END_DATA_BLOCK

DATA_BLOCK "IEC_Timer_0_DB_44"   // DB23
{ S7_Optimized_Access := 'TRUE' }
// stored: InstanceOfName IEC_TIMER, OfSystemLibElement IEC_TIMER, OfSystemLibVersion 1.0
"IEC_TIMER"
   // VAR
   //    PT : Time;
   //    ET { ExternalWritable := 'False'} : Time;
   //    IN : Bool;
   //    Q { ExternalWritable := 'False'} : Bool;
   // END_VAR
BEGIN
END_DATA_BLOCK

DATA_BLOCK "IEC_Timer_0_DB_45"   // DB30
{ S7_Optimized_Access := 'TRUE' }
// stored: InstanceOfName IEC_TIMER, OfSystemLibElement IEC_TIMER, OfSystemLibVersion 1.0
"IEC_TIMER"
   // VAR
   //    PT : Time;
   //    ET { ExternalWritable := 'False'} : Time;
   //    IN : Bool;
   //    Q { ExternalWritable := 'False'} : Bool;
   // END_VAR
BEGIN
END_DATA_BLOCK

DATA_BLOCK "IEC_Timer_0_DB_46"   // DB31
{ S7_Optimized_Access := 'TRUE' }
// stored: InstanceOfName IEC_TIMER, OfSystemLibElement IEC_TIMER, OfSystemLibVersion 1.0
"IEC_TIMER"
   // VAR
   //    PT : Time;
   //    ET { ExternalWritable := 'False'} : Time;
   //    IN : Bool;
   //    Q { ExternalWritable := 'False'} : Bool;
   // END_VAR
BEGIN
END_DATA_BLOCK

DATA_BLOCK "IEC_Timer_0_DB_5"   // DB46
{ S7_Optimized_Access := 'TRUE' }
// stored: InstanceOfName IEC_TIMER, OfSystemLibElement IEC_TIMER, OfSystemLibVersion 1.0
"IEC_TIMER"
   // VAR
   //    PT : Time;
   //    ET { ExternalWritable := 'False'} : Time;
   //    IN : Bool;
   //    Q { ExternalWritable := 'False'} : Bool;
   // END_VAR
BEGIN
END_DATA_BLOCK

DATA_BLOCK "IEC_Timer_0_DB_6"   // DB47
{ S7_Optimized_Access := 'TRUE' }
// stored: InstanceOfName IEC_TIMER, OfSystemLibElement IEC_TIMER, OfSystemLibVersion 1.0
"IEC_TIMER"
   // VAR
   //    PT : Time;
   //    ET { ExternalWritable := 'False'} : Time;
   //    IN : Bool;
   //    Q { ExternalWritable := 'False'} : Bool;
   // END_VAR
BEGIN
END_DATA_BLOCK

DATA_BLOCK "IEC_Timer_0_DB_7"   // DB49
{ S7_Optimized_Access := 'TRUE' }
// stored: InstanceOfName IEC_TIMER, OfSystemLibElement IEC_TIMER, OfSystemLibVersion 1.0
"IEC_TIMER"
   // VAR
   //    PT : Time;
   //    ET { ExternalWritable := 'False'} : Time;
   //    IN : Bool;
   //    Q { ExternalWritable := 'False'} : Bool;
   // END_VAR
BEGIN
END_DATA_BLOCK

DATA_BLOCK "IEC_Timer_0_DB_8"   // DB51
{ S7_Optimized_Access := 'TRUE' }
// stored: InstanceOfName IEC_TIMER, OfSystemLibElement IEC_TIMER, OfSystemLibVersion 1.0
"IEC_TIMER"
   // VAR
   //    PT : Time;
   //    ET { ExternalWritable := 'False'} : Time;
   //    IN : Bool;
   //    Q { ExternalWritable := 'False'} : Bool;
   // END_VAR
BEGIN
END_DATA_BLOCK

DATA_BLOCK "IEC_Timer_0_DB_9"   // DB53
{ S7_Optimized_Access := 'TRUE' }
// stored: InstanceOfName IEC_TIMER, OfSystemLibElement IEC_TIMER, OfSystemLibVersion 1.0
"IEC_TIMER"
   // VAR
   //    PT : Time;
   //    ET { ExternalWritable := 'False'} : Time;
   //    IN : Bool;
   //    Q { ExternalWritable := 'False'} : Bool;
   // END_VAR
BEGIN
END_DATA_BLOCK

DATA_BLOCK "IEC_Timer_0_DB_98"   // DB206
{ S7_Optimized_Access := 'TRUE' }
// stored: InstanceOfName IEC_TIMER, OfSystemLibElement IEC_TIMER, OfSystemLibVersion 1.0
"IEC_TIMER"
   // VAR
   //    PT : Time;
   //    ET { ExternalWritable := 'False'} : Time;
   //    IN : Bool;
   //    Q { ExternalWritable := 'False'} : Bool;
   // END_VAR
BEGIN
END_DATA_BLOCK

DATA_BLOCK "PID_PUMP_SPEED"   // DB85
// stored: InstanceOfName PID_Compact, OfSystemLibElement PID_Compact, OfSystemLibVersion 2.3
PID_Compact   // technology object, version 2.3
   // VAR_INPUT
   //    Setpoint : Real;
   //    Input : Real;
   //    Input_PER : Int;
   //    Disturbance : Real;
   //    ManualEnable : Bool;
   //    ManualValue : Real;
   //    ErrorAck : Bool;
   //    Reset : Bool;
   //    ModeActivate : Bool;
   // END_VAR
   // VAR_OUTPUT
   //    ScaledInput { ExternalWritable := 'False'} : Real;
   //    Output { ExternalWritable := 'False'} : Real;
   //    Output_PER { ExternalWritable := 'False'} : Int;
   //    Output_PWM { ExternalWritable := 'False'} : Bool;
   //    SetpointLimit_H { ExternalWritable := 'False'} : Bool;
   //    SetpointLimit_L { ExternalWritable := 'False'} : Bool;
   //    InputWarning_H { ExternalWritable := 'False'} : Bool;
   //    InputWarning_L { ExternalWritable := 'False'} : Bool;
   //    State { ExternalWritable := 'False'} : Int;
   //    Error { ExternalWritable := 'False'} : Bool;
   //    ErrorBits { ExternalWritable := 'False'} : DWord;
   // END_VAR
   // VAR_IN_OUT
   //    Mode : Int;
   // END_VAR
   // VAR
   //    InternalDiagnostic : DWord;
   //    InternalVersion { ExternalWritable := 'False'} : DWord;
   //    InternalRTVersion : DWord;
   //    IntegralResetMode { S7_SetPoint := 'True'} : Int;
   //    OverwriteInitialOutputValue : Real;
   //    RunModeByStartup { S7_SetPoint := 'True'} : Bool;
   //    LoadBackUp : Bool;
   //    SetSubstituteOutput { S7_SetPoint := 'True'} : Bool;
   //    PhysicalUnit { ExternalWritable := 'False'; S7_SetPoint := 'True'} : Int;
   //    PhysicalQuantity { ExternalWritable := 'False'; S7_SetPoint := 'True'} : Int;
   //    ActivateRecoverMode { S7_SetPoint := 'True'} : Bool;
   // END_VAR
   // VAR RETAIN
   //    Warning { ExternalWritable := 'False'} : DWord;
   //    WarningInternal { ExternalWritable := 'False'} : DWord;
   // END_VAR
   // VAR
   //    Progress { ExternalWritable := 'False'} : Real;
   //    CurrentSetpoint { ExternalWritable := 'False'} : Real;
   //    CancelTuningLevel { S7_SetPoint := 'True'} : Real;
   //    SubstituteOutput { S7_SetPoint := 'True'} : Real;
   //    Config { S7_SetPoint := 'True'} : PID_CompactConfig;
   //    CycleTime { S7_SetPoint := 'True'} : PID_CycleTime;
   //    CtrlParamsBackUp { S7_SetPoint := 'True'} : PID_CompactControlParams;
   //    PIDSelfTune { S7_SetPoint := 'True'} : PID_CompactSelfTune;
   //    PIDCtrl { S7_SetPoint := 'True'} : PID_CompactControl;
   // END_VAR
   // VAR RETAIN
   //    Retain { S7_SetPoint := 'True'} : PID_CompactRetain;
   // END_VAR
BEGIN
END_DATA_BLOCK
